FUNCTION_BLOCK fb_V3JRSModuleWithChiller
VAR_INPUT
	bBuiltInTemperetureController : BOOL;
	bBuiltInVacuumSensorController : BOOL;
	bBuiltInVacuumNegativeSignal : BOOL;
END_VAR
VAR_OUTPUT
END_VAR
VAR_IN_OUT
	DS_Alarm :DSV3_JRS_Alarm; (*Channel 200 ~ 204*)
	DS_HMI : DSV3_JRS_HMI; (*Channel of Other Digitial IO and DT*)
	DS_Input : DSV3_JRS_Input; (*Channel 0 ~ 3 *)
	DS_Output : DSV3_JRS_Output; (*Channel 100 ~ 103*)
END_VAR
VAR

	(*Analog Declaration*)
	iThermalOilTempAnalogInput			AT %I* : INT;
	iTopDistillatorTempAnalogInput			AT %I* : INT;
	iBottomDistillatorTempAnalogInput		AT %I* : INT;
	iVaporGenerationTempAnalogInput		AT %I* : INT;
	iColdWaterTankTempAnalogInput 		AT %I* : INT;

	iVacuumSensorAnalogInput				AT %I* : INT;



	(*AlarmControl*)
	arfbTimerAlarm: ARRAY [1..49] OF TIMER_ALARM;
	ARiBuzzerOut : ARRAY [1..4] OF INT;
	ARiAlarmFlag : ARRAY [1..4] OF INT;
	arCMP: ARRAY [1..32] OF CMP_OC_W1;


	(*Others*)
	EQGT: ARRAY [1..10] OF EQ_GT;


	tCompressorOnTimer: TON;
	tCompressorOffTimer: TON;
	tPowerOnDelayTimer: TON;
	tVaporGenTopUpDelayOff: TON;
	tThermalOilChangeResetPBTimer: TON;

	bPowerOnDelay: BOOL;

	t1SecCP: TON;

	tFreshHCCircPumpDelayOffTimer: TON;

	ARtAutoModeTimer: ARRAY [1..4] OF TON;
	ARtManualBoilingTimer: ARRAY [1..4] OF TON;
	diAutoModeDelayTimeSV_Sec: DINT := 20;

	bRecycleStartPBRE: R_TRIG;
	t1SecCPRE: R_TRIG;

	(*Auto BoilDown*)
	t570_AutoBoilingStartDelayTimer: TON;
	t571_AutoBoilDownCompletedDelayTimer: TON;
	t572_AutoBoilSludgeDrainCompletedDelayTimer: TON;
	t573_AutoBoilDistillatorDrainCompletedDelayTimer: TON;
	t574_AutoBoilSludgeDrainCoolingCompletedDelayTimer: TON;        (************* New extra request by customer - YCH************)

	bAutoBoilProcessCompletedFlag: BOOL;
	bAutoBoilDownCompletedFlag: BOOL;
	bAutoBoilSludgeDrainCompletedFlag: BOOL;
	bAutoBoilDistillatorDrainCompletedFlag: BOOL;
	bAutoBoilSludgeDrainCoolingCompletedFlag: BOOL;        (************* New extra request by customer - YCH************)

	(*Manual BoilDown*)
	t590_ManualBoilDownCompletedDelayTimer: TON;
	t591_ManualBoilSludgeCoolingCompletedDelayTimer: TON;
	t592_ManualBoilSludgeDrainCompletedDelayTimer: TON;
	bManualBoilDownCompletedFlag: BOOL;
	bManualBoilSludgeCoolingCompletedFlag: BOOL;
	bManualBoilSludgeDrainCompletedFlag: BOOL;
	bManualBoilSludgeDrainCompletedRE: R_TRIG;
	bManualBoilDownStartPBRE: R_TRIG;

	t592_ManualBoilSludgeDrainCompletedDelayTimerRE: R_TRIG;
	ARfbV2TempControl: ARRAY [1..5] OF fbV2_TempControl;
	rNIL: REAL;

	fbKeyenceVacSensorTuningkPa_Vacuum: fbKeyenceVacSensorTuningkPa;
	bVacuumAchieveFlag: BOOL;

	fbJRSMachine_Routine								: fbV2_EquipmentServiceCounter_Day;
	fbJRSMachine_Major									: fbV2_EquipmentServiceCounter_Day;

	bManulBoilPageOn:BOOL;
(*
	bInternalInput_b000_04_ThermalOilTempCtrlHighTempAlarmSignal : BOOL;
	bInternalInput_b000_05_ThermalOilTempCtrlReadySignal : BOOL;
	bInternalInput_b000_06_ThermalOilTempCtrlOnOffSignal : BOOL;
	bInternalInput_b000_04_ThermalOilTempCtrlHighTempAlarmSignal  : BOOL;
	bInternalInput_b000_05_ThermalOilTempCtrlReadySignal  : BOOL;
	bInternalInput_b000_06_ThermalOilTempCtrlOnOffSignal   : BOOL;

	bInternalInput_b000_07_TopDistillatorTempCtrlHighTempAlarmSignal : BOOL;
	bInternalInput_b000_08_TopDistillatorTempCtrlReadySignal : BOOL;
	bInternalInput_b000_09_TopDistillatorTempCtrlOnOffSignal : BOOL;
	bInternalInput_b000_07_TopDistillatorTempCtrlHighTempAlarmSignal  : BOOL;
	bInternalInput_b000_08_TopDistillatorTempCtrlReadySignal  : BOOL;
	bInternalInput_b000_09_TopDistillatorTempCtrlOnOffSignal   : BOOL;

	bInternalInput_b001_08_BottomDistillatorTempCtrlHighTempAlarmSignal : BOOL;
	bInternalInput_b001_09_BottomDistillatorTempCtrlReadySignal : BOOL;
	bInternalInput_b001_10_BottomDistillatorTempCtrlOnOffSignal : BOOL;
	bInternalInput_b001_08_BottomDistillatorTempCtrlHighTempAlarmSignal  : BOOL;
	bInternalInput_b001_09_BottomDistillatorTempCtrlReadySignal  : BOOL;
	bInternalInput_b001_10_BottomDistillatorTempCtrlOnOffSignal   : BOOL;

	bInternalInput_b002_00_VaporGenerationTempCtrlHighTempAlarmSignal : BOOL;
	bInternalInput_b002_01_VaporGenerationTempCtrlReadySignal : BOOL;
	bInternalInput_b002_02_VaporGenerationTempCtrlOnOffSignal : BOOL;
	bInternalInput_b002_00_VaporGenerationTempCtrlHighTempAlarmSignal  : BOOL;
	bInternalInput_b002_01_VaporGenerationTempCtrlReadySignal  : BOOL;
	bInternalInput_b002_02_VaporGenerationTempCtrlOnOffSignal  : BOOL;


	bInternalInput_b003_03_ColdWaterTankTempCtrlHighTempAlarmSignal : BOOL;
	bInternalInput_b003_04_ColdWaterTankTempCtrlReadySignal : BOOL;
	bInternalInput_b003_05_ColdWaterTankTempCtrlOnOffSignal	 : BOOL;
	bInternalInput_b003_03_ColdWaterTankTempCtrlHighTempAlarmSignal  : BOOL;
	bInternalInput_b003_04_ColdWaterTankTempCtrlReadySignal  : BOOL;
	bInternalInput_b003_05_ColdWaterTankTempCtrlOnOffSignal  : BOOL;

	bInternalInput_b001_04_VacuumNotAchieveSignal	: BOOL;
	bInternalInput_b001_04_VacuumNotAchieveSignal  : BOOL;

*)

	(*Internal Signal Declaration*)
	bInternalAlarm_b200_00_FreshHCTankCircPumpTORAlarm   : BOOL;
	bInternalAlarm_b200_01_CircTankCircPumpTORAlarm   : BOOL;
	bInternalAlarm_b200_02_ThermalOilPumpTORAlarm   : BOOL;
	bInternalAlarm_b200_03_ThermalOilLowLevelAlarm   : BOOL;
	bInternalAlarm_b200_04_ThermalOilTempHighAlarm   : BOOL;
	bInternalAlarm_b200_05_ThermalOilTempNotReadyAlarm   : BOOL;
	bInternalAlarm_b200_06_ThermalOilHeaterOnOffAlarm   : BOOL;
	bInternalAlarm_b200_07_TopDistillatorTempHighAlarm   : BOOL;
	bInternalAlarm_b200_08_TopDistillatorTempNotReadyAlarm   : BOOL;
	bInternalAlarm_b200_09_TopDistillatorHeaterOnOffAlarm   : BOOL;
	bInternalAlarm_b200_10_RecycleStartStopPBAlarm   : BOOL;
	bInternalAlarm_b200_11_EstopPBAlarm   : BOOL;

	bInternalAlarm_b201_00_PhaseSeqenceRelayAlarm   : BOOL;
	bInternalAlarm_b201_01_ThermalOilUpThermostatAlarm   : BOOL;
	bInternalAlarm_b201_02_SludgeTankHighLevelAlarm   : BOOL;
	bInternalAlarm_b201_03_FreshHCTankLowLevelAlarm   : BOOL;
	bInternalAlarm_b201_04_VacuumNotAchieveAlarm   : BOOL;
	bInternalAlarm_b201_05_IncomingCDALowPressureAlarm   : BOOL;
	bInternalAlarm_b201_06_CoolingWaterLowFlowAlarm   : BOOL;
	bInternalAlarm_b201_07_CircularTankLowLevelAlarm   : BOOL;
	bInternalAlarm_b201_08_BottomDistillatorTempHighAlarm   : BOOL;
	bInternalAlarm_b201_09_BottomDistillatorTempNotReadyAlarm   : BOOL;
	bInternalAlarm_b201_10_BottomDistillatorHeaterOnOffAlarm   : BOOL;
	bInternalAlarm_b201_11_ThermalOilDownThermostatAlarm   : BOOL;
	bInternalAlarm_b201_12_ThermalOilMidThermostatAlarm   : BOOL;

	bInternalAlarm_b202_00_VaporGenerationTempHighAlarm   : BOOL;
	bInternalAlarm_b202_01_VaporGenerationTempNotReadyAlarm   : BOOL;
	bInternalAlarm_b202_02_VaporGenerationHeaterOnOffAlarm   : BOOL;
	bInternalAlarm_b202_03_WasteCollectionTankLowLevelAlarm   : BOOL;
	bInternalAlarm_b202_04_VaporGenerationTankLowLevelAlarm   : BOOL;
	bInternalAlarm_b202_05_HCPurgingAV3_1Alarm   : BOOL;
	bInternalAlarm_b202_06_MainMachineWasteTankLowLevelAlarm   : BOOL;
	bInternalAlarm_b202_07_MainMachineWasteTankHighLevelAlarm   : BOOL;
	bInternalAlarm_b202_08_ReservedAlarm   : BOOL;
	bInternalAlarm_b202_09_ReservedAlarm   : BOOL;
	bInternalAlarm_b202_10_ReservedAlarm   : BOOL;
	bInternalAlarm_b202_11_ReservedAlarm   : BOOL;

	bInternalAlarm_b203_00_ChillerSelectorOnOffAlarm   : BOOL;
	bInternalAlarm_b203_01_ColdWaterTankLowLevelAlarm   : BOOL;
	bInternalAlarm_b203_02_SludgeTankMissingAlarm   : BOOL;
	bInternalAlarm_b203_03_ColdWaterTankTempHighAlarm   : BOOL;
	bInternalAlarm_b203_04_ColdWaterTankTempNotReadyAlarm   : BOOL;
	bInternalAlarm_b203_05_ColdWaterTankHeaterOnOffAlarm   : BOOL;
	bInternalAlarm_b203_06_ChillerPumpTORAlarm   : BOOL;
	bInternalAlarm_b203_07_ChillerFlowSwitchAlarm   : BOOL;
	bInternalAlarm_b203_08_ChillerInterlockRelayAlarm   : BOOL;
	bInternalAlarm_b203_09_ReservedAlarm   : BOOL;
	bInternalAlarm_b203_10_ThermalOilChangeWarning   : BOOL;
	bInternalAlarm_b203_11_ThermalOilChangeAlarm   : BOOL;



	bInternalInput_b000_00_FreshHCTankCircPumpTOR   : BOOL;
	bInternalInput_b000_01_CircTankCircPumpTOR   : BOOL;
	bInternalInput_b000_02_ThermalOilPumpTOR  : BOOL;
	bInternalInput_b000_03_ThermalOilLevelSensor  : BOOL;
	bInternalInput_b000_04_ThermalOilTempCtrlHighTempAlarmSignal  : BOOL;
	bInternalInput_b000_05_ThermalOilTempCtrlReadySignal  : BOOL;
	bInternalInput_b000_06_ThermalOilTempCtrlOnOffSignal   : BOOL;
	bInternalInput_b000_07_TopDistillatorTempCtrlHighTempAlarmSignal  : BOOL;
	bInternalInput_b000_08_TopDistillatorTempCtrlReadySignal  : BOOL;
	bInternalInput_b000_09_TopDistillatorTempCtrlOnOffSignal   : BOOL;
	bInternalInput_b000_10_RecycleStartStopPB  : BOOL;
	bInternalInput_b000_11_EStopPB  : BOOL;


	bInternalInput_b001_00_PhaseSequenceRelayAlarm  : BOOL;
	bInternalInput_b001_01_ThermalOilUpThermostat   : BOOL;
	bInternalInput_b001_02_SludgeTankLevelSensor  : BOOL;
	bInternalInput_b001_03_FreshHCTankLevelSensor  : BOOL;
	bInternalInput_b001_04_VacuumNotAchieveSignal  : BOOL;
	bInternalInput_b001_05_IncomingCDAPressureSwitch  : BOOL;
	bInternalInput_b001_06_CoolingWaterFlowSwitch  : BOOL;
	bInternalInput_b001_07_CircularTankLevelSensor  : BOOL;
	bInternalInput_b001_08_BottomDistillatorTempCtrlHighTempAlarmSignal  : BOOL;
	bInternalInput_b001_09_BottomDistillatorTempCtrlReadySignal  : BOOL;
	bInternalInput_b001_10_BottomDistillatorTempCtrlOnOffSignal   : BOOL;
	bInternalInput_b001_11_ThermalOilDownThermostat  : BOOL;
	bInternalInput_b001_12_ThermalOilMidThermostat  : BOOL;

	bInternalInput_b002_00_VaporGenerationTempCtrlHighTempAlarmSignal  : BOOL;
	bInternalInput_b002_01_VaporGenerationTempCtrlReadySignal  : BOOL;
	bInternalInput_b002_02_VaporGenerationTempCtrlOnOffSignal  : BOOL;
	bInternalInput_b002_03_WasteCollectionTankLevelSensor  : BOOL;
	bInternalInput_b002_04_VaporGenerationTankLowLevelSensor  : BOOL;
	bInternalInput_b002_05_HCPurgingAV  : BOOL;
	bInternalInput_b002_06_MainMachineWasteCollectTankLowLevelSignal  : BOOL;
	bInternalInput_b002_07_MainMachineWasteCollectTankHighLevelSignal  : BOOL;
	bInternalInput_b002_08_FromMainMachineSignal3  : BOOL;
	bInternalInput_b002_09_FromMainMachineSignal4  : BOOL;
	bInternalInput_b002_10_FromMainMachineSignal5  : BOOL;
	bInternalInput_b002_11_ReservedAlarmSignal  : BOOL;


	bInternalInput_b003_00_ChillerSelectorOnOff  : BOOL;
	bInternalInput_b003_01_ColdWaterTankLowLevelSensor  : BOOL;
	bInternalInput_b003_02_SludgeTankPresentSensor  : BOOL;
	bInternalInput_b003_03_ColdWaterTankTempCtrlHighTempAlarmSignal  : BOOL;
	bInternalInput_b003_04_ColdWaterTankTempCtrlReadySignal  : BOOL;
	bInternalInput_b003_05_ColdWaterTankTempCtrlOnOffSignal  : BOOL;
	bInternalInput_b003_06_ChillerPumpTOR  : BOOL;
	bInternalInput_b003_07_ChillerFlowSwitch  : BOOL;
	bInternalInput_b003_08_ChillerInterlockRelay  : BOOL;
	bInternalInput_b003_09_ReservedAlarmSignal  : BOOL;
	bInternalInput_b003_10_ReservedAlarmSignal  : BOOL;
	bInternalInput_b003_11_ReservedAlarmSignal  : BOOL;


	bInternalOutput_b100_00_FreshHCTankCircPumpOnOff   : BOOL;
	bInternalOutput_b100_01_CircTankCircPumpOnOff  : BOOL;
	bInternalOutput_b100_02_ThermalOilPumpOnOff  : BOOL;
	bInternalOutput_b100_03_ThermalOilHeaterOnOff  : BOOL;
	bInternalOutput_b100_04_Buzzer  : BOOL;
	bInternalOutput_b100_05_RecycleStartStopIndicator  : BOOL;
	bInternalOutput_b100_06_Reserved  : BOOL;
	bInternalOutput_b100_07_UFOVacuumRelease32WayAV  : BOOL;


	bInternalOutput_b101_00_CondenserTankVacuumReleaseAV  : BOOL;
	bInternalOutput_b101_01_WasteSludgeCollectionDrumAV   : BOOL;
	bInternalOutput_b101_02_DistillationTankDrainAV  : BOOL;
	bInternalOutput_b101_03_EconomizerAV  : BOOL;
	bInternalOutput_b101_04_Reserved  : BOOL;
	bInternalOutput_b101_05_Reserved  : BOOL;
	bInternalOutput_b101_06_VaporGenerationAV  : BOOL;
	bInternalOutput_b101_07_VacuumSharingAV  : BOOL;


	bInternalOutput_b102_00_RecycleReadySignal  : BOOL;
	bInternalOutput_b102_01_VaporNotAvailableForRequestSignal  : BOOL;
	bInternalOutput_b102_02_ToMainMachineSignal3  : BOOL;
	bInternalOutput_b102_03_ToMainMachineSignal4  : BOOL;
	bInternalOutput_b102_04_ToMainMachineSignal5  : BOOL;
	bInternalOutput_b102_05_Reserved  : BOOL;
	bInternalOutput_b102_06_Reserved  : BOOL;
	bInternalOutput_b102_07_Reserved  : BOOL;


	bInternalOutput_b103_00_ChillerPumpOnOff  : BOOL;
	bInternalOutput_b103_01_Reserved  : BOOL;
	bInternalOutput_b103_02_Reserved  : BOOL;
	bInternalOutput_b103_03_Reserved  : BOOL;
	bInternalOutput_b103_04_ChillerSelectorOnOffIndicator  : BOOL;
	bInternalOutput_b103_05_ChillerReadySignal  : BOOL;
	bInternalOutput_b103_06_ChillerCompressorOnOff  : BOOL;
	bInternalOutput_b103_07_Reserved  : BOOL;


END_VAR
VAR // added by the converter: edge detectors and wires of the graphical bodies
    _w1, _w3, _w4, _w5, _w6, _w7, _w8, _w9 : ANY;
    _w2 : BOOL;
END_VAR

	(*Timer*)
	t1SecCP(IN:=NOT t1SecCP.Q , PT:=t#1s , Q=> , ET=> );


	(*R_TRIG*)
	t1SecCPRE(CLK:=t1SecCP.Q , Q=> );
	bRecycleStartPBRE(CLK:=bInternalInput_b000_10_RecycleStartStopPB , Q=> );


	(*Sub Program Execution*)
	Z_Mapping();
	Other_LD();
	Other_ST();
	FixOutput_LD();
	OutputCtrl_LD();
	AlarmCtrl_LD();
	BuzzerCtrl_ST();
	MessageDisplayCtrl_ST();
	AutoHCTopUp_LD();
	HighLowLimitCtrl_ST();
	AutoCtrl_LD();
	ManualCtrl_ST();
	
	AutoBoilingCtrl_LD();
	AutoBoilingCtrl_ST();

	ManualBoilingCtrl_LD();
	ManualBoilingCtrl_ST();


	ThermalOilChangeHRMeter_ST();
	ChillerCtrl_LD();
	SystemRestore_LD();
	Z_BuiltInTempCtrl_ST();

	Z_BuiltInVacuumCtrl_ST();

	JRSMachineServiceCtrl_LD();

ACTION AlarmCtrl_LD:
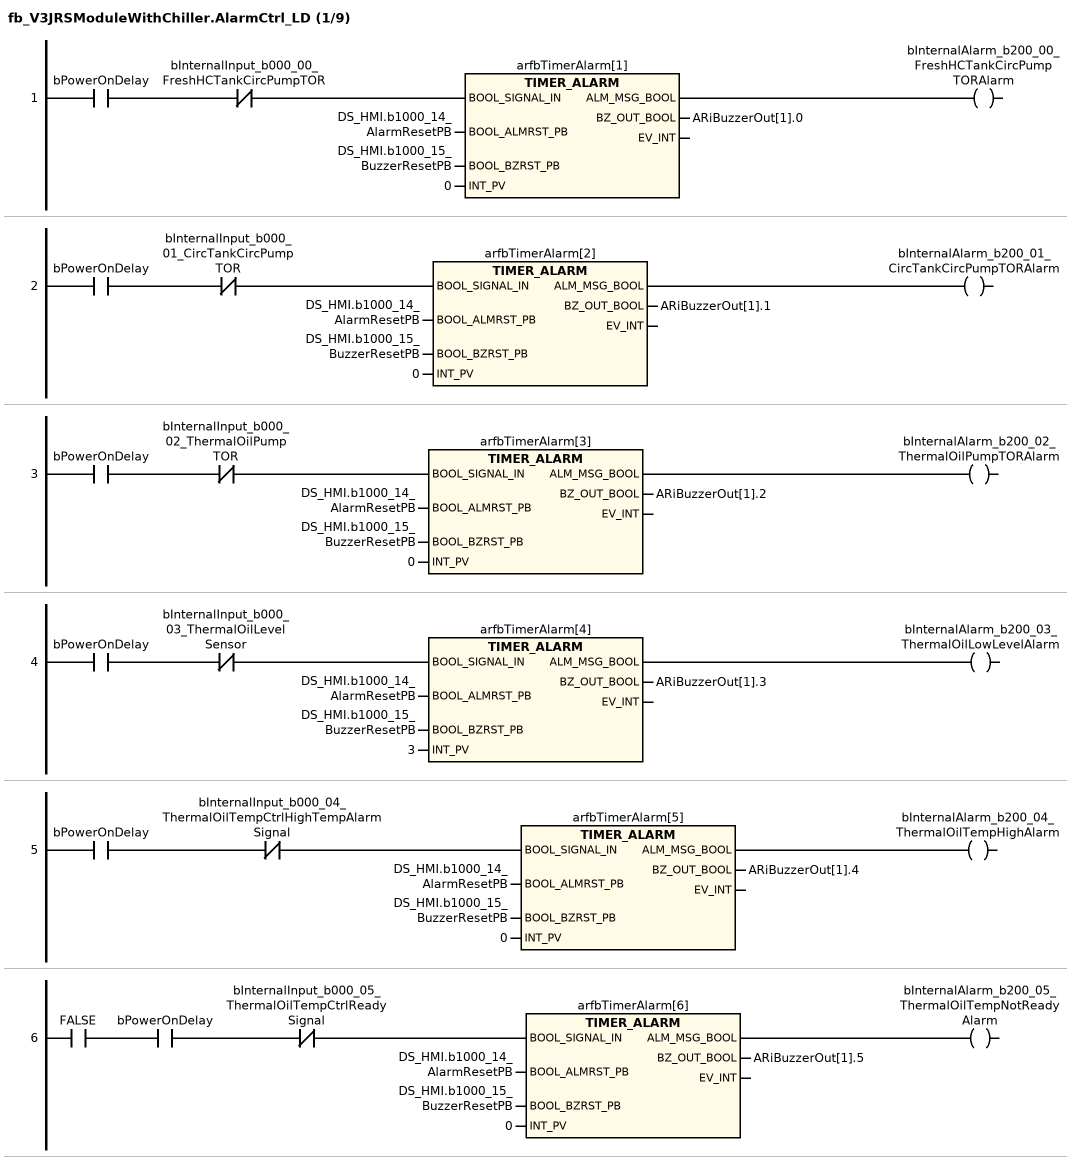
// NETWORK 1
arfbTimerAlarm[1](
    BOOL_SIGNAL_IN := bPowerOnDelay AND NOT bInternalInput_b000_00_FreshHCTankCircPumpTOR,
    BOOL_ALMRST_PB := DS_HMI.b1000_14_AlarmResetPB,
    BOOL_BZRST_PB := DS_HMI.b1000_15_BuzzerResetPB,
    INT_PV := 0,
    BZ_OUT_BOOL => ARiBuzzerOut[1].0); // TIMER_ALARM
bInternalAlarm_b200_00_FreshHCTankCircPumpTORAlarm := arfbTimerAlarm[1].ALM_MSG_BOOL;

// NETWORK 2
arfbTimerAlarm[2](
    BOOL_SIGNAL_IN := bPowerOnDelay AND NOT bInternalInput_b000_01_CircTankCircPumpTOR,
    BOOL_ALMRST_PB := DS_HMI.b1000_14_AlarmResetPB,
    BOOL_BZRST_PB := DS_HMI.b1000_15_BuzzerResetPB,
    INT_PV := 0,
    BZ_OUT_BOOL => ARiBuzzerOut[1].1); // TIMER_ALARM
bInternalAlarm_b200_01_CircTankCircPumpTORAlarm := arfbTimerAlarm[2].ALM_MSG_BOOL;

// NETWORK 3
arfbTimerAlarm[3](
    BOOL_SIGNAL_IN := bPowerOnDelay AND NOT bInternalInput_b000_02_ThermalOilPumpTOR,
    BOOL_ALMRST_PB := DS_HMI.b1000_14_AlarmResetPB,
    BOOL_BZRST_PB := DS_HMI.b1000_15_BuzzerResetPB,
    INT_PV := 0,
    BZ_OUT_BOOL => ARiBuzzerOut[1].2); // TIMER_ALARM
bInternalAlarm_b200_02_ThermalOilPumpTORAlarm := arfbTimerAlarm[3].ALM_MSG_BOOL;

// NETWORK 4
arfbTimerAlarm[4](
    BOOL_SIGNAL_IN := bPowerOnDelay AND NOT bInternalInput_b000_03_ThermalOilLevelSensor,
    BOOL_ALMRST_PB := DS_HMI.b1000_14_AlarmResetPB,
    BOOL_BZRST_PB := DS_HMI.b1000_15_BuzzerResetPB,
    INT_PV := 3,
    BZ_OUT_BOOL => ARiBuzzerOut[1].3); // TIMER_ALARM
bInternalAlarm_b200_03_ThermalOilLowLevelAlarm := arfbTimerAlarm[4].ALM_MSG_BOOL;

// NETWORK 5
arfbTimerAlarm[5](
    BOOL_SIGNAL_IN := bPowerOnDelay AND NOT bInternalInput_b000_04_ThermalOilTempCtrlHighTempAlarmSignal,
    BOOL_ALMRST_PB := DS_HMI.b1000_14_AlarmResetPB,
    BOOL_BZRST_PB := DS_HMI.b1000_15_BuzzerResetPB,
    INT_PV := 0,
    BZ_OUT_BOOL => ARiBuzzerOut[1].4); // TIMER_ALARM
bInternalAlarm_b200_04_ThermalOilTempHighAlarm := arfbTimerAlarm[5].ALM_MSG_BOOL;

// NETWORK 6
arfbTimerAlarm[6](
    BOOL_SIGNAL_IN := FALSE AND bPowerOnDelay AND NOT bInternalInput_b000_05_ThermalOilTempCtrlReadySignal,
    BOOL_ALMRST_PB := DS_HMI.b1000_14_AlarmResetPB,
    BOOL_BZRST_PB := DS_HMI.b1000_15_BuzzerResetPB,
    INT_PV := 0,
    BZ_OUT_BOOL => ARiBuzzerOut[1].5); // TIMER_ALARM
bInternalAlarm_b200_05_ThermalOilTempNotReadyAlarm := arfbTimerAlarm[6].ALM_MSG_BOOL;

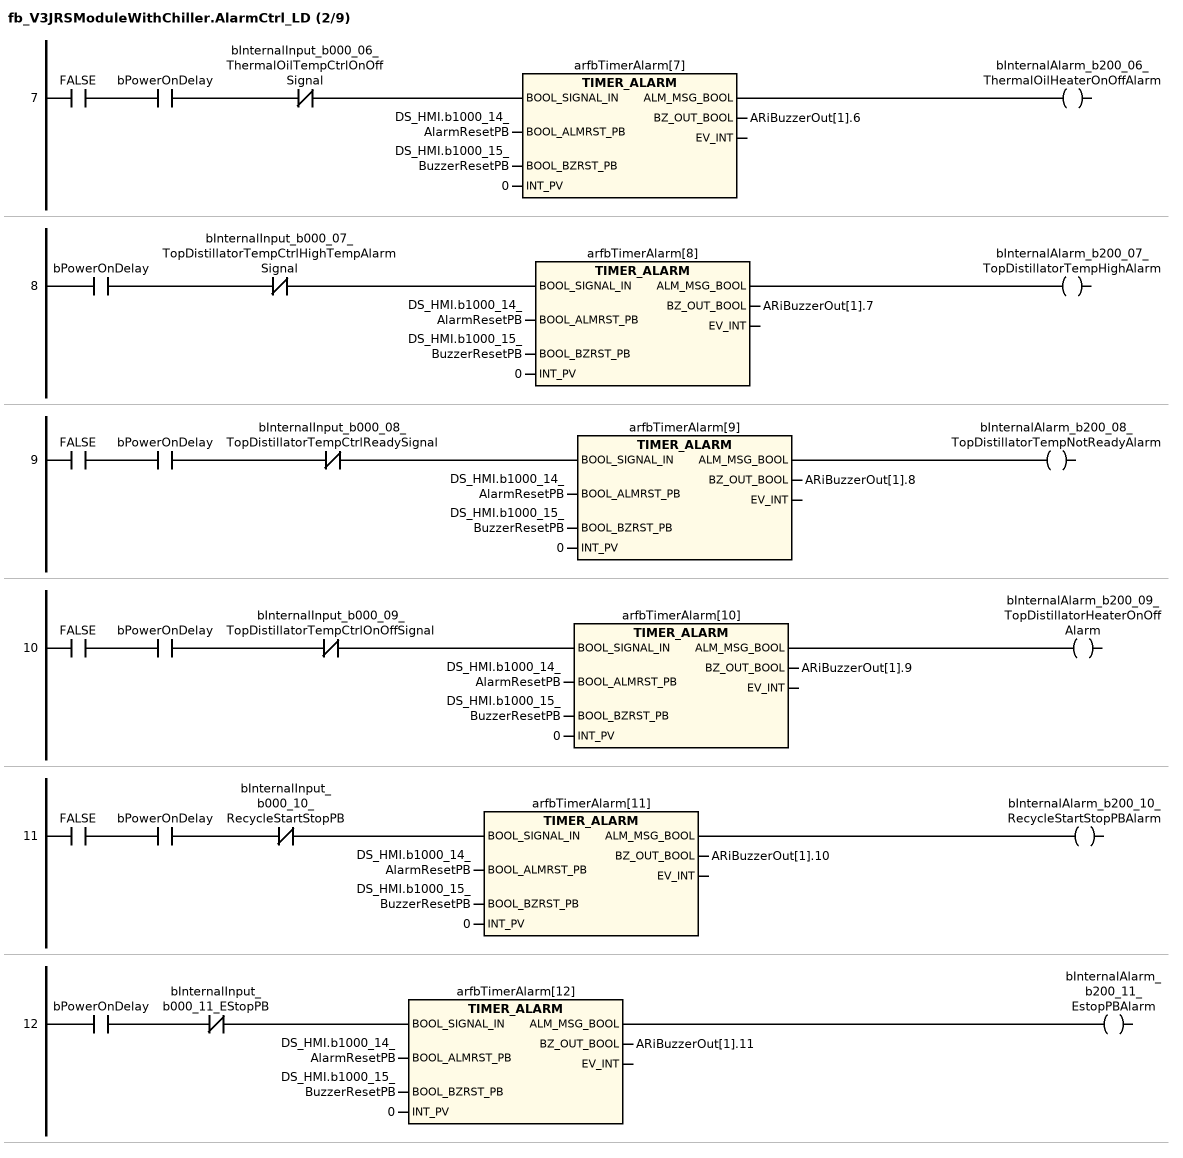
// NETWORK 7
arfbTimerAlarm[7](
    BOOL_SIGNAL_IN := FALSE AND bPowerOnDelay AND NOT bInternalInput_b000_06_ThermalOilTempCtrlOnOffSignal,
    BOOL_ALMRST_PB := DS_HMI.b1000_14_AlarmResetPB,
    BOOL_BZRST_PB := DS_HMI.b1000_15_BuzzerResetPB,
    INT_PV := 0,
    BZ_OUT_BOOL => ARiBuzzerOut[1].6); // TIMER_ALARM
bInternalAlarm_b200_06_ThermalOilHeaterOnOffAlarm := arfbTimerAlarm[7].ALM_MSG_BOOL;

// NETWORK 8
arfbTimerAlarm[8](
    BOOL_SIGNAL_IN := bPowerOnDelay AND NOT bInternalInput_b000_07_TopDistillatorTempCtrlHighTempAlarmSignal,
    BOOL_ALMRST_PB := DS_HMI.b1000_14_AlarmResetPB,
    BOOL_BZRST_PB := DS_HMI.b1000_15_BuzzerResetPB,
    INT_PV := 0,
    BZ_OUT_BOOL => ARiBuzzerOut[1].7); // TIMER_ALARM
bInternalAlarm_b200_07_TopDistillatorTempHighAlarm := arfbTimerAlarm[8].ALM_MSG_BOOL;

// NETWORK 9
arfbTimerAlarm[9](
    BOOL_SIGNAL_IN := FALSE AND bPowerOnDelay AND NOT bInternalInput_b000_08_TopDistillatorTempCtrlReadySignal,
    BOOL_ALMRST_PB := DS_HMI.b1000_14_AlarmResetPB,
    BOOL_BZRST_PB := DS_HMI.b1000_15_BuzzerResetPB,
    INT_PV := 0,
    BZ_OUT_BOOL => ARiBuzzerOut[1].8); // TIMER_ALARM
bInternalAlarm_b200_08_TopDistillatorTempNotReadyAlarm := arfbTimerAlarm[9].ALM_MSG_BOOL;

// NETWORK 10
arfbTimerAlarm[10](
    BOOL_SIGNAL_IN := FALSE AND bPowerOnDelay AND NOT bInternalInput_b000_09_TopDistillatorTempCtrlOnOffSignal,
    BOOL_ALMRST_PB := DS_HMI.b1000_14_AlarmResetPB,
    BOOL_BZRST_PB := DS_HMI.b1000_15_BuzzerResetPB,
    INT_PV := 0,
    BZ_OUT_BOOL => ARiBuzzerOut[1].9); // TIMER_ALARM
bInternalAlarm_b200_09_TopDistillatorHeaterOnOffAlarm := arfbTimerAlarm[10].ALM_MSG_BOOL;

// NETWORK 11
arfbTimerAlarm[11](
    BOOL_SIGNAL_IN := FALSE AND bPowerOnDelay AND NOT bInternalInput_b000_10_RecycleStartStopPB,
    BOOL_ALMRST_PB := DS_HMI.b1000_14_AlarmResetPB,
    BOOL_BZRST_PB := DS_HMI.b1000_15_BuzzerResetPB,
    INT_PV := 0,
    BZ_OUT_BOOL => ARiBuzzerOut[1].10); // TIMER_ALARM
bInternalAlarm_b200_10_RecycleStartStopPBAlarm := arfbTimerAlarm[11].ALM_MSG_BOOL;

// NETWORK 12
arfbTimerAlarm[12](
    BOOL_SIGNAL_IN := bPowerOnDelay AND NOT bInternalInput_b000_11_EStopPB,
    BOOL_ALMRST_PB := DS_HMI.b1000_14_AlarmResetPB,
    BOOL_BZRST_PB := DS_HMI.b1000_15_BuzzerResetPB,
    INT_PV := 0,
    BZ_OUT_BOOL => ARiBuzzerOut[1].11); // TIMER_ALARM
bInternalAlarm_b200_11_EstopPBAlarm := arfbTimerAlarm[12].ALM_MSG_BOOL;

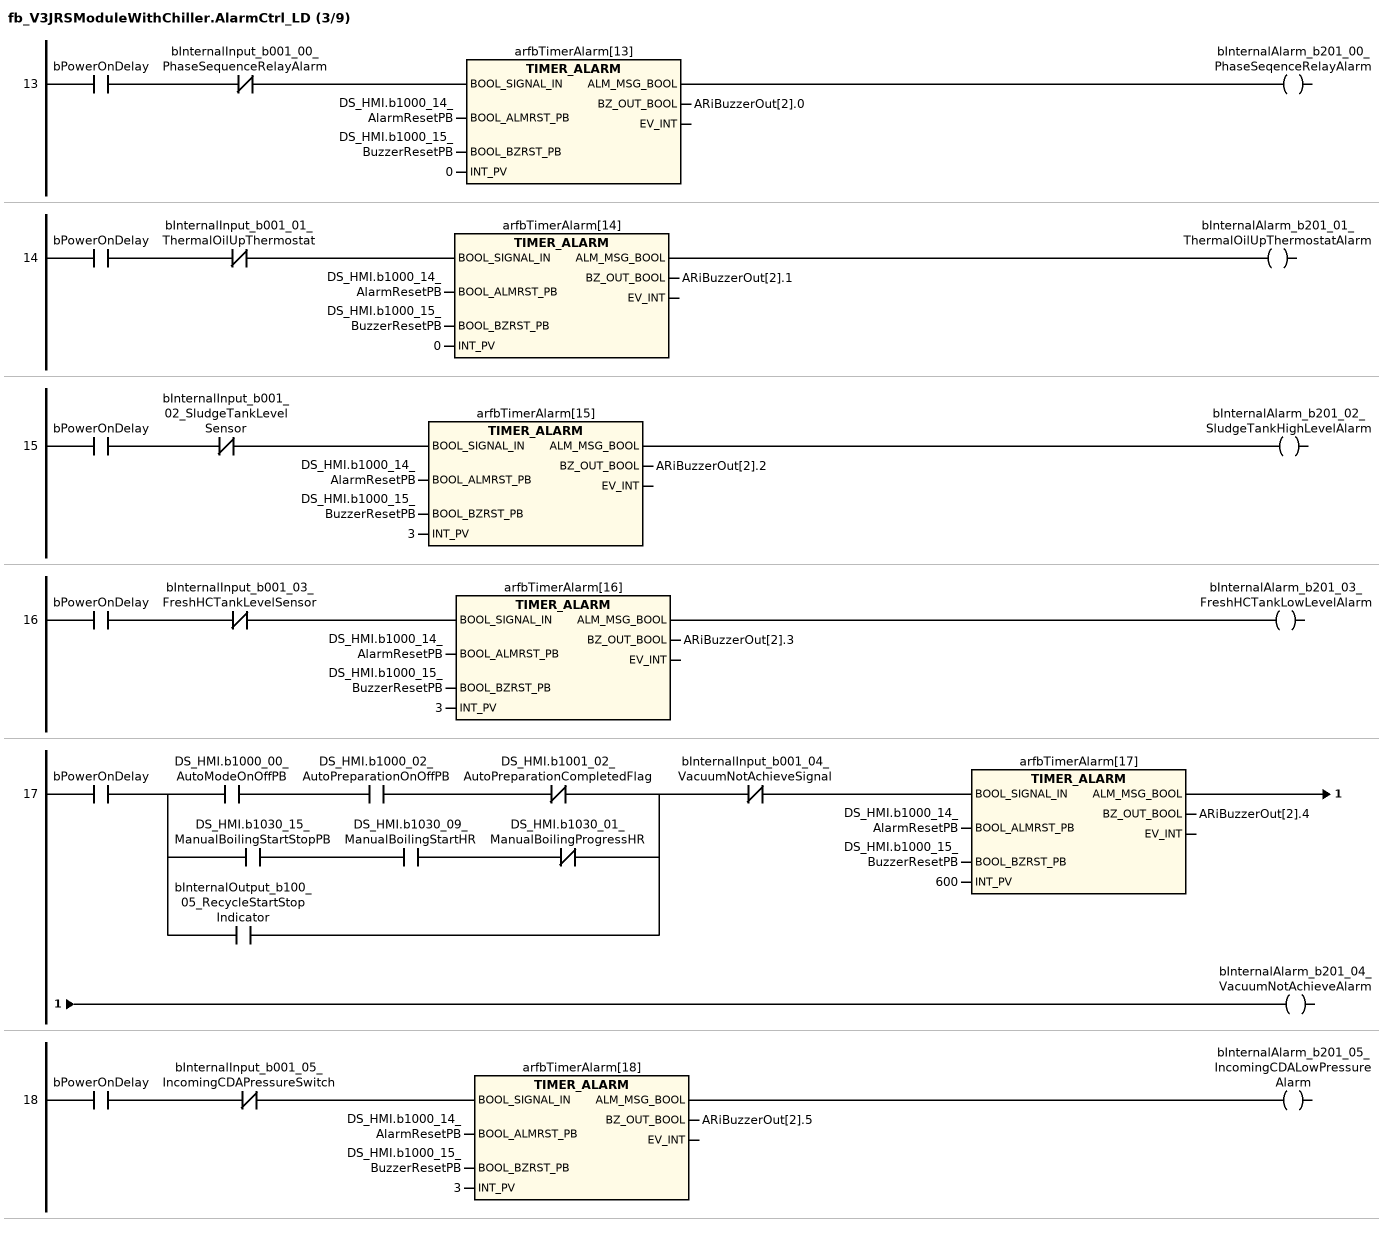
// NETWORK 13
arfbTimerAlarm[13](
    BOOL_SIGNAL_IN := bPowerOnDelay AND NOT bInternalInput_b001_00_PhaseSequenceRelayAlarm,
    BOOL_ALMRST_PB := DS_HMI.b1000_14_AlarmResetPB,
    BOOL_BZRST_PB := DS_HMI.b1000_15_BuzzerResetPB,
    INT_PV := 0,
    BZ_OUT_BOOL => ARiBuzzerOut[2].0); // TIMER_ALARM
bInternalAlarm_b201_00_PhaseSeqenceRelayAlarm := arfbTimerAlarm[13].ALM_MSG_BOOL;

// NETWORK 14
arfbTimerAlarm[14](
    BOOL_SIGNAL_IN := bPowerOnDelay AND NOT bInternalInput_b001_01_ThermalOilUpThermostat,
    BOOL_ALMRST_PB := DS_HMI.b1000_14_AlarmResetPB,
    BOOL_BZRST_PB := DS_HMI.b1000_15_BuzzerResetPB,
    INT_PV := 0,
    BZ_OUT_BOOL => ARiBuzzerOut[2].1); // TIMER_ALARM
bInternalAlarm_b201_01_ThermalOilUpThermostatAlarm := arfbTimerAlarm[14].ALM_MSG_BOOL;

// NETWORK 15
arfbTimerAlarm[15](
    BOOL_SIGNAL_IN := bPowerOnDelay AND NOT bInternalInput_b001_02_SludgeTankLevelSensor,
    BOOL_ALMRST_PB := DS_HMI.b1000_14_AlarmResetPB,
    BOOL_BZRST_PB := DS_HMI.b1000_15_BuzzerResetPB,
    INT_PV := 3,
    BZ_OUT_BOOL => ARiBuzzerOut[2].2); // TIMER_ALARM
bInternalAlarm_b201_02_SludgeTankHighLevelAlarm := arfbTimerAlarm[15].ALM_MSG_BOOL;

// NETWORK 16
arfbTimerAlarm[16](
    BOOL_SIGNAL_IN := bPowerOnDelay AND NOT bInternalInput_b001_03_FreshHCTankLevelSensor,
    BOOL_ALMRST_PB := DS_HMI.b1000_14_AlarmResetPB,
    BOOL_BZRST_PB := DS_HMI.b1000_15_BuzzerResetPB,
    INT_PV := 3,
    BZ_OUT_BOOL => ARiBuzzerOut[2].3); // TIMER_ALARM
bInternalAlarm_b201_03_FreshHCTankLowLevelAlarm := arfbTimerAlarm[16].ALM_MSG_BOOL;

// NETWORK 17
arfbTimerAlarm[17](
    BOOL_SIGNAL_IN := (bPowerOnDelay AND (DS_HMI.b1000_00_AutoModeOnOffPB AND DS_HMI.b1000_02_AutoPreparationOnOffPB AND NOT DS_HMI.b1001_02_AutoPreparationCompletedFlag OR DS_HMI.b1030_15_ManualBoilingStartStopPB AND DS_HMI.b1030_09_ManualBoilingStartHR AND NOT DS_HMI.b1030_01_ManualBoilingProgressHR OR bInternalOutput_b100_05_RecycleStartStopIndicator)) AND NOT bInternalInput_b001_04_VacuumNotAchieveSignal,
    BOOL_ALMRST_PB := DS_HMI.b1000_14_AlarmResetPB,
    BOOL_BZRST_PB := DS_HMI.b1000_15_BuzzerResetPB,
    INT_PV := 600,
    BZ_OUT_BOOL => ARiBuzzerOut[2].4); // TIMER_ALARM
bInternalAlarm_b201_04_VacuumNotAchieveAlarm := arfbTimerAlarm[17].ALM_MSG_BOOL;

// NETWORK 18
arfbTimerAlarm[18](
    BOOL_SIGNAL_IN := bPowerOnDelay AND NOT bInternalInput_b001_05_IncomingCDAPressureSwitch,
    BOOL_ALMRST_PB := DS_HMI.b1000_14_AlarmResetPB,
    BOOL_BZRST_PB := DS_HMI.b1000_15_BuzzerResetPB,
    INT_PV := 3,
    BZ_OUT_BOOL => ARiBuzzerOut[2].5); // TIMER_ALARM
bInternalAlarm_b201_05_IncomingCDALowPressureAlarm := arfbTimerAlarm[18].ALM_MSG_BOOL;

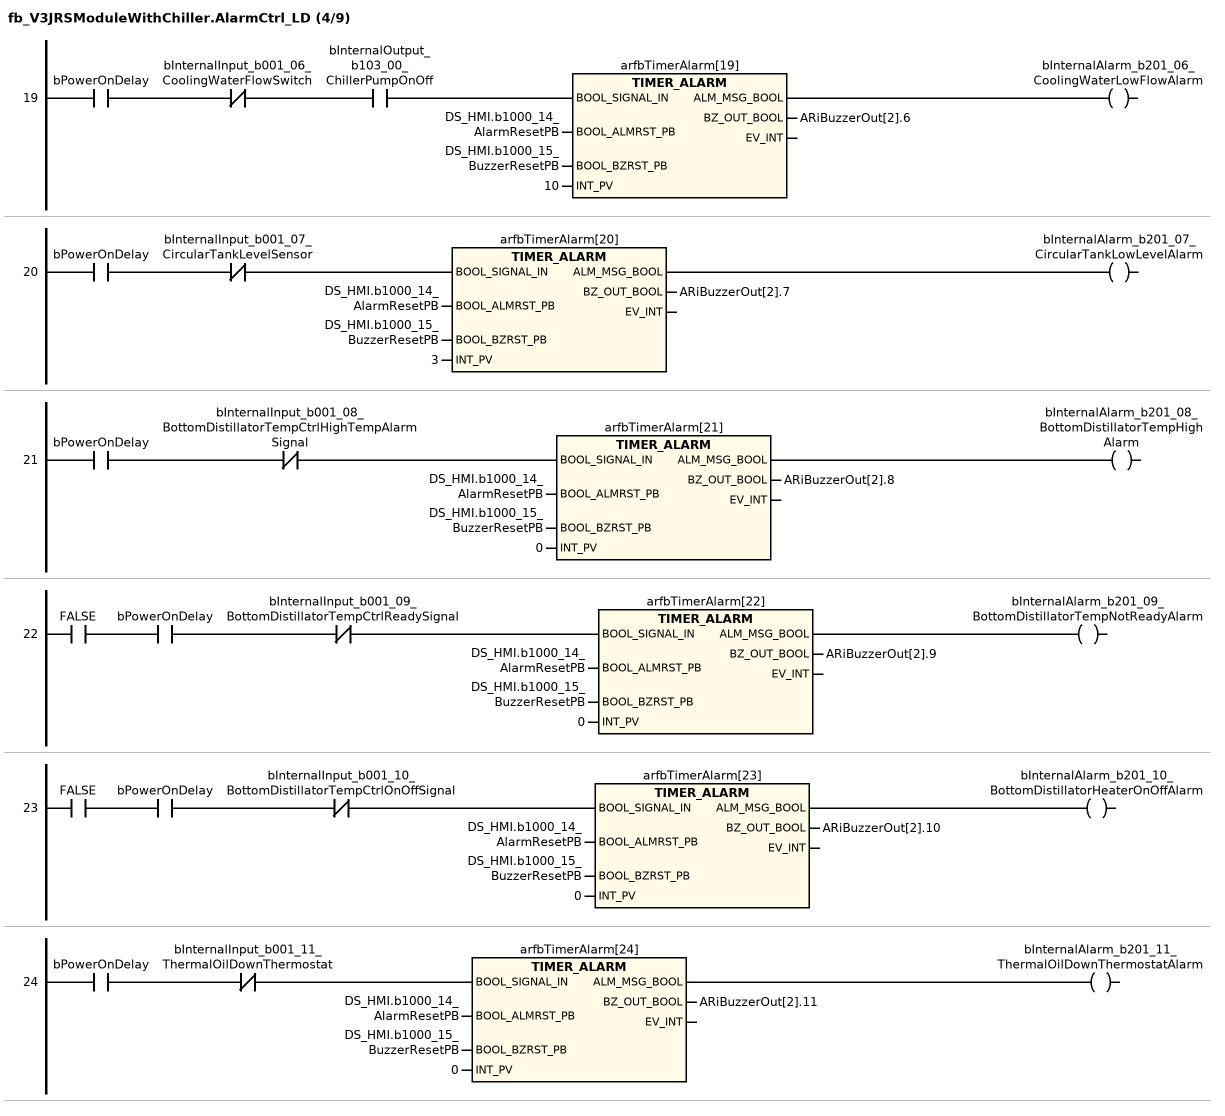
// NETWORK 19
arfbTimerAlarm[19](
    BOOL_SIGNAL_IN := bPowerOnDelay AND NOT bInternalInput_b001_06_CoolingWaterFlowSwitch AND bInternalOutput_b103_00_ChillerPumpOnOff,
    BOOL_ALMRST_PB := DS_HMI.b1000_14_AlarmResetPB,
    BOOL_BZRST_PB := DS_HMI.b1000_15_BuzzerResetPB,
    INT_PV := 10,
    BZ_OUT_BOOL => ARiBuzzerOut[2].6); // TIMER_ALARM
bInternalAlarm_b201_06_CoolingWaterLowFlowAlarm := arfbTimerAlarm[19].ALM_MSG_BOOL;

// NETWORK 20
arfbTimerAlarm[20](
    BOOL_SIGNAL_IN := bPowerOnDelay AND NOT bInternalInput_b001_07_CircularTankLevelSensor,
    BOOL_ALMRST_PB := DS_HMI.b1000_14_AlarmResetPB,
    BOOL_BZRST_PB := DS_HMI.b1000_15_BuzzerResetPB,
    INT_PV := 3,
    BZ_OUT_BOOL => ARiBuzzerOut[2].7); // TIMER_ALARM
bInternalAlarm_b201_07_CircularTankLowLevelAlarm := arfbTimerAlarm[20].ALM_MSG_BOOL;

// NETWORK 21
arfbTimerAlarm[21](
    BOOL_SIGNAL_IN := bPowerOnDelay AND NOT bInternalInput_b001_08_BottomDistillatorTempCtrlHighTempAlarmSignal,
    BOOL_ALMRST_PB := DS_HMI.b1000_14_AlarmResetPB,
    BOOL_BZRST_PB := DS_HMI.b1000_15_BuzzerResetPB,
    INT_PV := 0,
    BZ_OUT_BOOL => ARiBuzzerOut[2].8); // TIMER_ALARM
bInternalAlarm_b201_08_BottomDistillatorTempHighAlarm := arfbTimerAlarm[21].ALM_MSG_BOOL;

// NETWORK 22
arfbTimerAlarm[22](
    BOOL_SIGNAL_IN := FALSE AND bPowerOnDelay AND NOT bInternalInput_b001_09_BottomDistillatorTempCtrlReadySignal,
    BOOL_ALMRST_PB := DS_HMI.b1000_14_AlarmResetPB,
    BOOL_BZRST_PB := DS_HMI.b1000_15_BuzzerResetPB,
    INT_PV := 0,
    BZ_OUT_BOOL => ARiBuzzerOut[2].9); // TIMER_ALARM
bInternalAlarm_b201_09_BottomDistillatorTempNotReadyAlarm := arfbTimerAlarm[22].ALM_MSG_BOOL;

// NETWORK 23
arfbTimerAlarm[23](
    BOOL_SIGNAL_IN := FALSE AND bPowerOnDelay AND NOT bInternalInput_b001_10_BottomDistillatorTempCtrlOnOffSignal,
    BOOL_ALMRST_PB := DS_HMI.b1000_14_AlarmResetPB,
    BOOL_BZRST_PB := DS_HMI.b1000_15_BuzzerResetPB,
    INT_PV := 0,
    BZ_OUT_BOOL => ARiBuzzerOut[2].10); // TIMER_ALARM
bInternalAlarm_b201_10_BottomDistillatorHeaterOnOffAlarm := arfbTimerAlarm[23].ALM_MSG_BOOL;

// NETWORK 24
arfbTimerAlarm[24](
    BOOL_SIGNAL_IN := bPowerOnDelay AND NOT bInternalInput_b001_11_ThermalOilDownThermostat,
    BOOL_ALMRST_PB := DS_HMI.b1000_14_AlarmResetPB,
    BOOL_BZRST_PB := DS_HMI.b1000_15_BuzzerResetPB,
    INT_PV := 0,
    BZ_OUT_BOOL => ARiBuzzerOut[2].11); // TIMER_ALARM
bInternalAlarm_b201_11_ThermalOilDownThermostatAlarm := arfbTimerAlarm[24].ALM_MSG_BOOL;

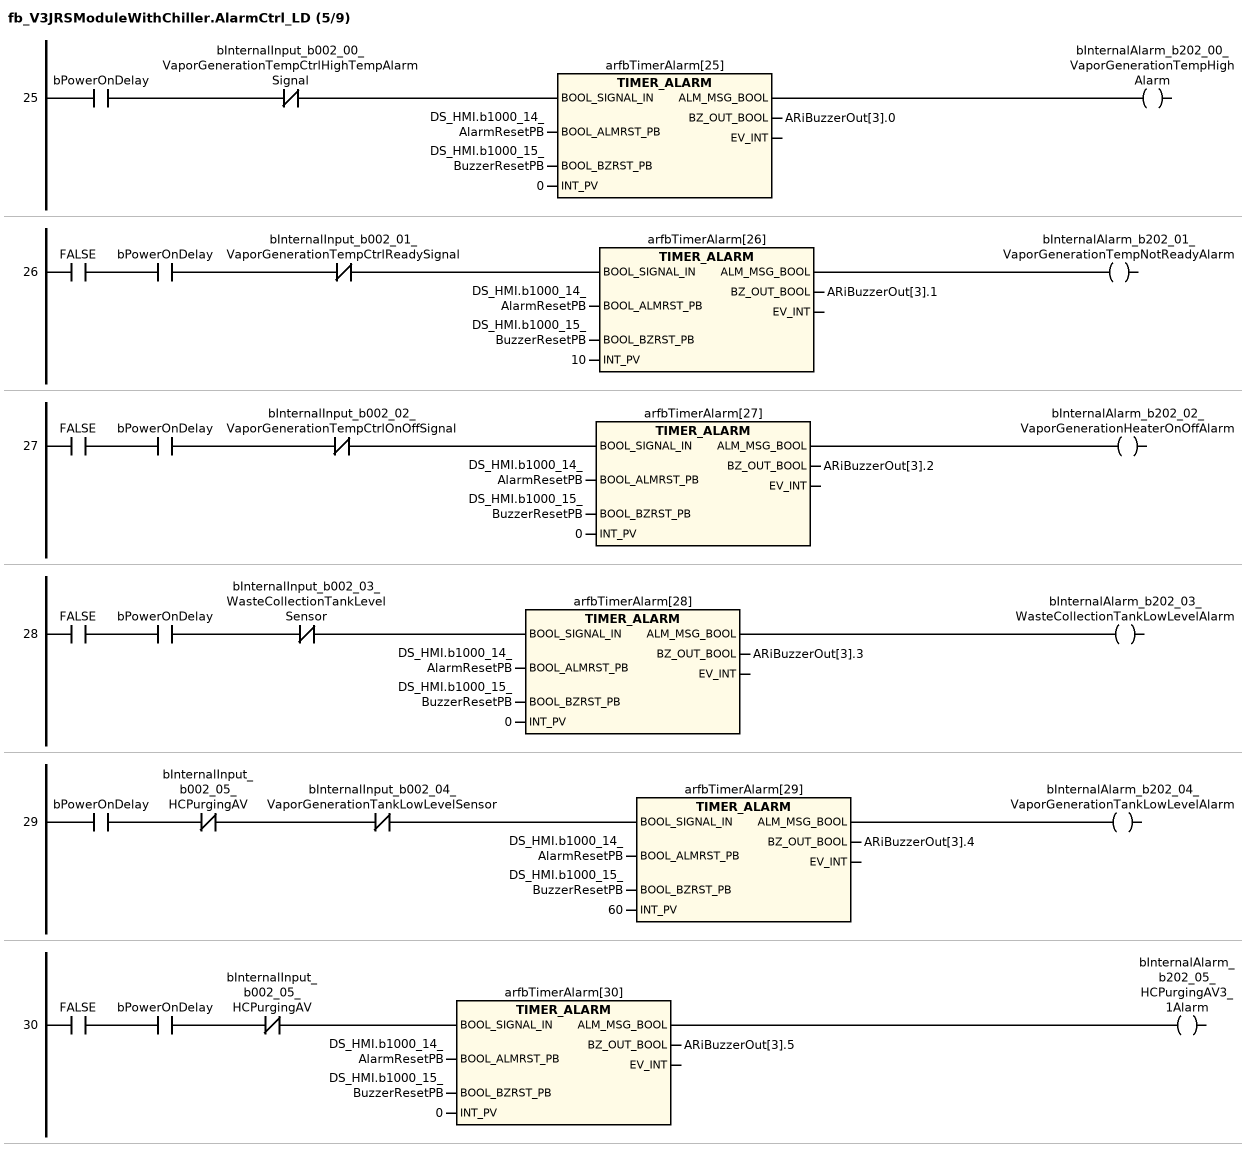
// NETWORK 25
arfbTimerAlarm[25](
    BOOL_SIGNAL_IN := bPowerOnDelay AND NOT bInternalInput_b002_00_VaporGenerationTempCtrlHighTempAlarmSignal,
    BOOL_ALMRST_PB := DS_HMI.b1000_14_AlarmResetPB,
    BOOL_BZRST_PB := DS_HMI.b1000_15_BuzzerResetPB,
    INT_PV := 0,
    BZ_OUT_BOOL => ARiBuzzerOut[3].0); // TIMER_ALARM
bInternalAlarm_b202_00_VaporGenerationTempHighAlarm := arfbTimerAlarm[25].ALM_MSG_BOOL;

// NETWORK 26
arfbTimerAlarm[26](
    BOOL_SIGNAL_IN := FALSE AND bPowerOnDelay AND NOT bInternalInput_b002_01_VaporGenerationTempCtrlReadySignal,
    BOOL_ALMRST_PB := DS_HMI.b1000_14_AlarmResetPB,
    BOOL_BZRST_PB := DS_HMI.b1000_15_BuzzerResetPB,
    INT_PV := 10,
    BZ_OUT_BOOL => ARiBuzzerOut[3].1); // TIMER_ALARM
bInternalAlarm_b202_01_VaporGenerationTempNotReadyAlarm := arfbTimerAlarm[26].ALM_MSG_BOOL;

// NETWORK 27
arfbTimerAlarm[27](
    BOOL_SIGNAL_IN := FALSE AND bPowerOnDelay AND NOT bInternalInput_b002_02_VaporGenerationTempCtrlOnOffSignal,
    BOOL_ALMRST_PB := DS_HMI.b1000_14_AlarmResetPB,
    BOOL_BZRST_PB := DS_HMI.b1000_15_BuzzerResetPB,
    INT_PV := 0,
    BZ_OUT_BOOL => ARiBuzzerOut[3].2); // TIMER_ALARM
bInternalAlarm_b202_02_VaporGenerationHeaterOnOffAlarm := arfbTimerAlarm[27].ALM_MSG_BOOL;

// NETWORK 28
arfbTimerAlarm[28](
    BOOL_SIGNAL_IN := FALSE AND bPowerOnDelay AND NOT bInternalInput_b002_03_WasteCollectionTankLevelSensor,
    BOOL_ALMRST_PB := DS_HMI.b1000_14_AlarmResetPB,
    BOOL_BZRST_PB := DS_HMI.b1000_15_BuzzerResetPB,
    INT_PV := 0,
    BZ_OUT_BOOL => ARiBuzzerOut[3].3); // TIMER_ALARM
bInternalAlarm_b202_03_WasteCollectionTankLowLevelAlarm := arfbTimerAlarm[28].ALM_MSG_BOOL;

// NETWORK 29
arfbTimerAlarm[29](
    BOOL_SIGNAL_IN := bPowerOnDelay AND NOT bInternalInput_b002_05_HCPurgingAV AND NOT bInternalInput_b002_04_VaporGenerationTankLowLevelSensor,
    BOOL_ALMRST_PB := DS_HMI.b1000_14_AlarmResetPB,
    BOOL_BZRST_PB := DS_HMI.b1000_15_BuzzerResetPB,
    INT_PV := 60,
    BZ_OUT_BOOL => ARiBuzzerOut[3].4); // TIMER_ALARM
bInternalAlarm_b202_04_VaporGenerationTankLowLevelAlarm := arfbTimerAlarm[29].ALM_MSG_BOOL;

// NETWORK 30
arfbTimerAlarm[30](
    BOOL_SIGNAL_IN := FALSE AND bPowerOnDelay AND NOT bInternalInput_b002_05_HCPurgingAV,
    BOOL_ALMRST_PB := DS_HMI.b1000_14_AlarmResetPB,
    BOOL_BZRST_PB := DS_HMI.b1000_15_BuzzerResetPB,
    INT_PV := 0,
    BZ_OUT_BOOL => ARiBuzzerOut[3].5); // TIMER_ALARM
bInternalAlarm_b202_05_HCPurgingAV3_1Alarm := arfbTimerAlarm[30].ALM_MSG_BOOL;

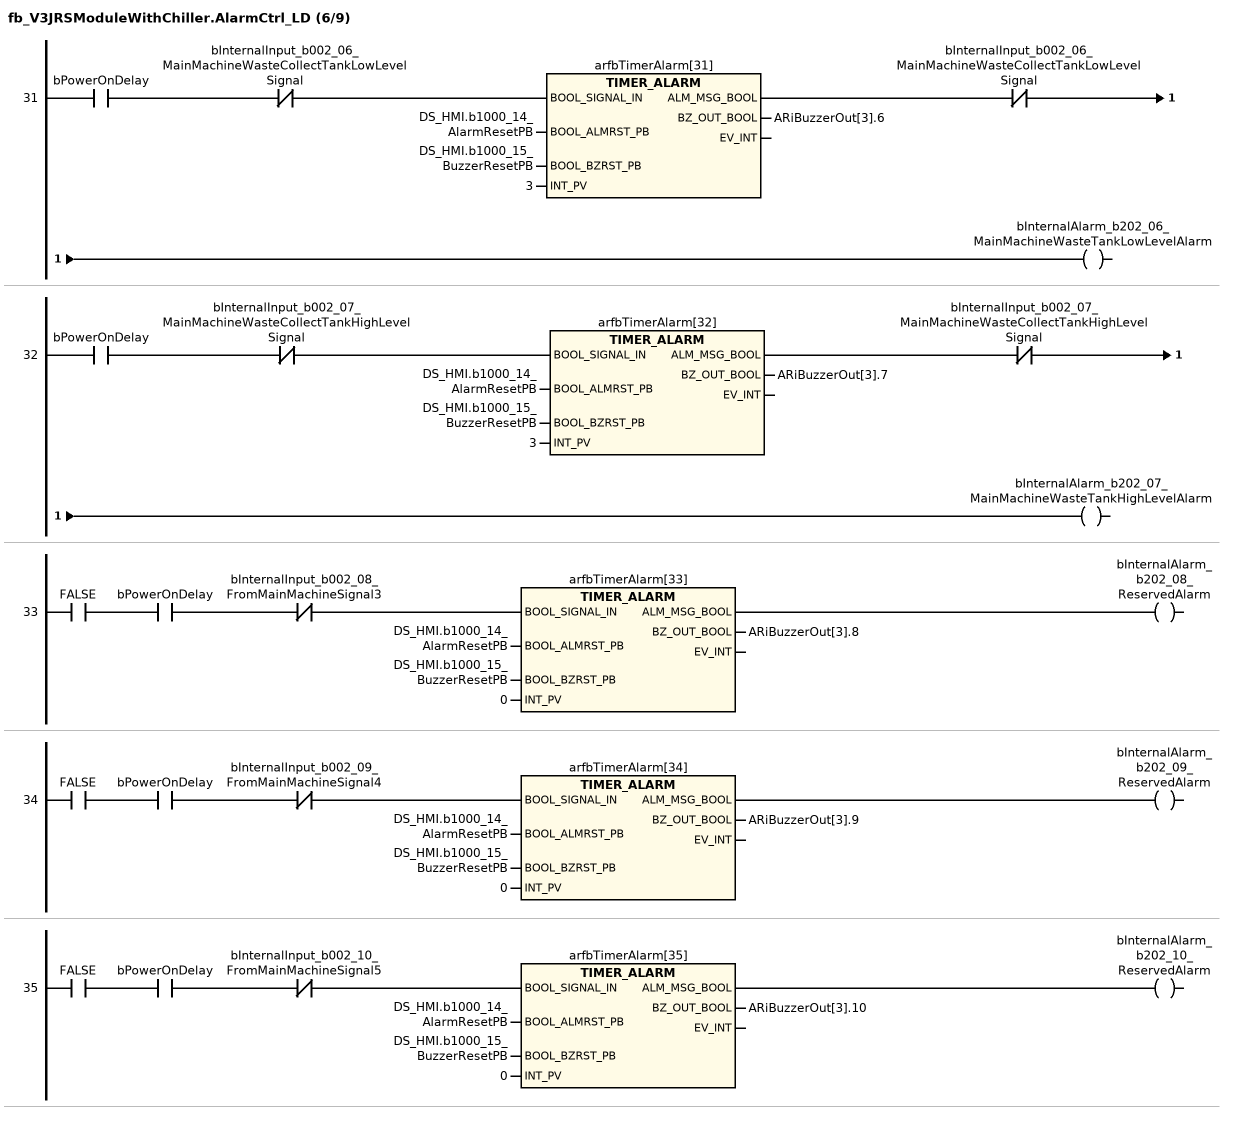
// NETWORK 31
arfbTimerAlarm[31](
    BOOL_SIGNAL_IN := bPowerOnDelay AND NOT bInternalInput_b002_06_MainMachineWasteCollectTankLowLevelSignal,
    BOOL_ALMRST_PB := DS_HMI.b1000_14_AlarmResetPB,
    BOOL_BZRST_PB := DS_HMI.b1000_15_BuzzerResetPB,
    INT_PV := 3,
    BZ_OUT_BOOL => ARiBuzzerOut[3].6); // TIMER_ALARM
bInternalAlarm_b202_06_MainMachineWasteTankLowLevelAlarm := arfbTimerAlarm[31].ALM_MSG_BOOL AND NOT bInternalInput_b002_06_MainMachineWasteCollectTankLowLevelSignal;

// NETWORK 32
arfbTimerAlarm[32](
    BOOL_SIGNAL_IN := bPowerOnDelay AND NOT bInternalInput_b002_07_MainMachineWasteCollectTankHighLevelSignal,
    BOOL_ALMRST_PB := DS_HMI.b1000_14_AlarmResetPB,
    BOOL_BZRST_PB := DS_HMI.b1000_15_BuzzerResetPB,
    INT_PV := 3,
    BZ_OUT_BOOL => ARiBuzzerOut[3].7); // TIMER_ALARM
bInternalAlarm_b202_07_MainMachineWasteTankHighLevelAlarm := arfbTimerAlarm[32].ALM_MSG_BOOL AND NOT bInternalInput_b002_07_MainMachineWasteCollectTankHighLevelSignal;

// NETWORK 33
arfbTimerAlarm[33](
    BOOL_SIGNAL_IN := FALSE AND bPowerOnDelay AND NOT bInternalInput_b002_08_FromMainMachineSignal3,
    BOOL_ALMRST_PB := DS_HMI.b1000_14_AlarmResetPB,
    BOOL_BZRST_PB := DS_HMI.b1000_15_BuzzerResetPB,
    INT_PV := 0,
    BZ_OUT_BOOL => ARiBuzzerOut[3].8); // TIMER_ALARM
bInternalAlarm_b202_08_ReservedAlarm := arfbTimerAlarm[33].ALM_MSG_BOOL;

// NETWORK 34
arfbTimerAlarm[34](
    BOOL_SIGNAL_IN := FALSE AND bPowerOnDelay AND NOT bInternalInput_b002_09_FromMainMachineSignal4,
    BOOL_ALMRST_PB := DS_HMI.b1000_14_AlarmResetPB,
    BOOL_BZRST_PB := DS_HMI.b1000_15_BuzzerResetPB,
    INT_PV := 0,
    BZ_OUT_BOOL => ARiBuzzerOut[3].9); // TIMER_ALARM
bInternalAlarm_b202_09_ReservedAlarm := arfbTimerAlarm[34].ALM_MSG_BOOL;

// NETWORK 35
arfbTimerAlarm[35](
    BOOL_SIGNAL_IN := FALSE AND bPowerOnDelay AND NOT bInternalInput_b002_10_FromMainMachineSignal5,
    BOOL_ALMRST_PB := DS_HMI.b1000_14_AlarmResetPB,
    BOOL_BZRST_PB := DS_HMI.b1000_15_BuzzerResetPB,
    INT_PV := 0,
    BZ_OUT_BOOL => ARiBuzzerOut[3].10); // TIMER_ALARM
bInternalAlarm_b202_10_ReservedAlarm := arfbTimerAlarm[35].ALM_MSG_BOOL;

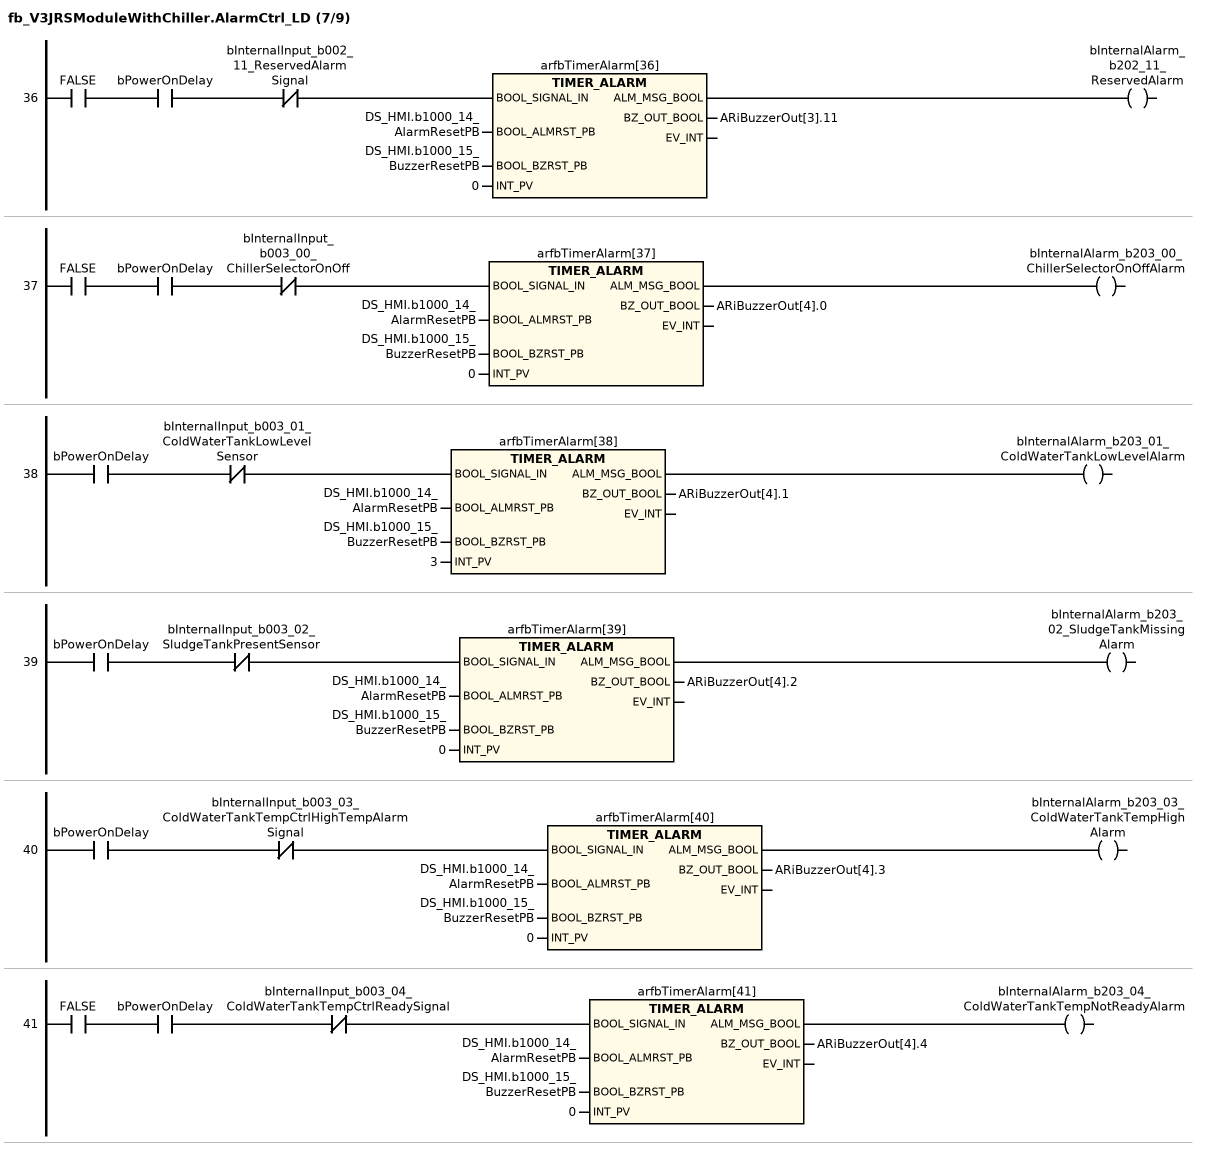
// NETWORK 36
arfbTimerAlarm[36](
    BOOL_SIGNAL_IN := FALSE AND bPowerOnDelay AND NOT bInternalInput_b002_11_ReservedAlarmSignal,
    BOOL_ALMRST_PB := DS_HMI.b1000_14_AlarmResetPB,
    BOOL_BZRST_PB := DS_HMI.b1000_15_BuzzerResetPB,
    INT_PV := 0,
    BZ_OUT_BOOL => ARiBuzzerOut[3].11); // TIMER_ALARM
bInternalAlarm_b202_11_ReservedAlarm := arfbTimerAlarm[36].ALM_MSG_BOOL;

// NETWORK 37
arfbTimerAlarm[37](
    BOOL_SIGNAL_IN := FALSE AND bPowerOnDelay AND NOT bInternalInput_b003_00_ChillerSelectorOnOff,
    BOOL_ALMRST_PB := DS_HMI.b1000_14_AlarmResetPB,
    BOOL_BZRST_PB := DS_HMI.b1000_15_BuzzerResetPB,
    INT_PV := 0,
    BZ_OUT_BOOL => ARiBuzzerOut[4].0); // TIMER_ALARM
bInternalAlarm_b203_00_ChillerSelectorOnOffAlarm := arfbTimerAlarm[37].ALM_MSG_BOOL;

// NETWORK 38
arfbTimerAlarm[38](
    BOOL_SIGNAL_IN := bPowerOnDelay AND NOT bInternalInput_b003_01_ColdWaterTankLowLevelSensor,
    BOOL_ALMRST_PB := DS_HMI.b1000_14_AlarmResetPB,
    BOOL_BZRST_PB := DS_HMI.b1000_15_BuzzerResetPB,
    INT_PV := 3,
    BZ_OUT_BOOL => ARiBuzzerOut[4].1); // TIMER_ALARM
bInternalAlarm_b203_01_ColdWaterTankLowLevelAlarm := arfbTimerAlarm[38].ALM_MSG_BOOL;

// NETWORK 39
arfbTimerAlarm[39](
    BOOL_SIGNAL_IN := bPowerOnDelay AND NOT bInternalInput_b003_02_SludgeTankPresentSensor,
    BOOL_ALMRST_PB := DS_HMI.b1000_14_AlarmResetPB,
    BOOL_BZRST_PB := DS_HMI.b1000_15_BuzzerResetPB,
    INT_PV := 0,
    BZ_OUT_BOOL => ARiBuzzerOut[4].2); // TIMER_ALARM
bInternalAlarm_b203_02_SludgeTankMissingAlarm := arfbTimerAlarm[39].ALM_MSG_BOOL;

// NETWORK 40
arfbTimerAlarm[40](
    BOOL_SIGNAL_IN := bPowerOnDelay AND NOT bInternalInput_b003_03_ColdWaterTankTempCtrlHighTempAlarmSignal,
    BOOL_ALMRST_PB := DS_HMI.b1000_14_AlarmResetPB,
    BOOL_BZRST_PB := DS_HMI.b1000_15_BuzzerResetPB,
    INT_PV := 0,
    BZ_OUT_BOOL => ARiBuzzerOut[4].3); // TIMER_ALARM
bInternalAlarm_b203_03_ColdWaterTankTempHighAlarm := arfbTimerAlarm[40].ALM_MSG_BOOL;

// NETWORK 41
arfbTimerAlarm[41](
    BOOL_SIGNAL_IN := FALSE AND bPowerOnDelay AND NOT bInternalInput_b003_04_ColdWaterTankTempCtrlReadySignal,
    BOOL_ALMRST_PB := DS_HMI.b1000_14_AlarmResetPB,
    BOOL_BZRST_PB := DS_HMI.b1000_15_BuzzerResetPB,
    INT_PV := 0,
    BZ_OUT_BOOL => ARiBuzzerOut[4].4); // TIMER_ALARM
bInternalAlarm_b203_04_ColdWaterTankTempNotReadyAlarm := arfbTimerAlarm[41].ALM_MSG_BOOL;

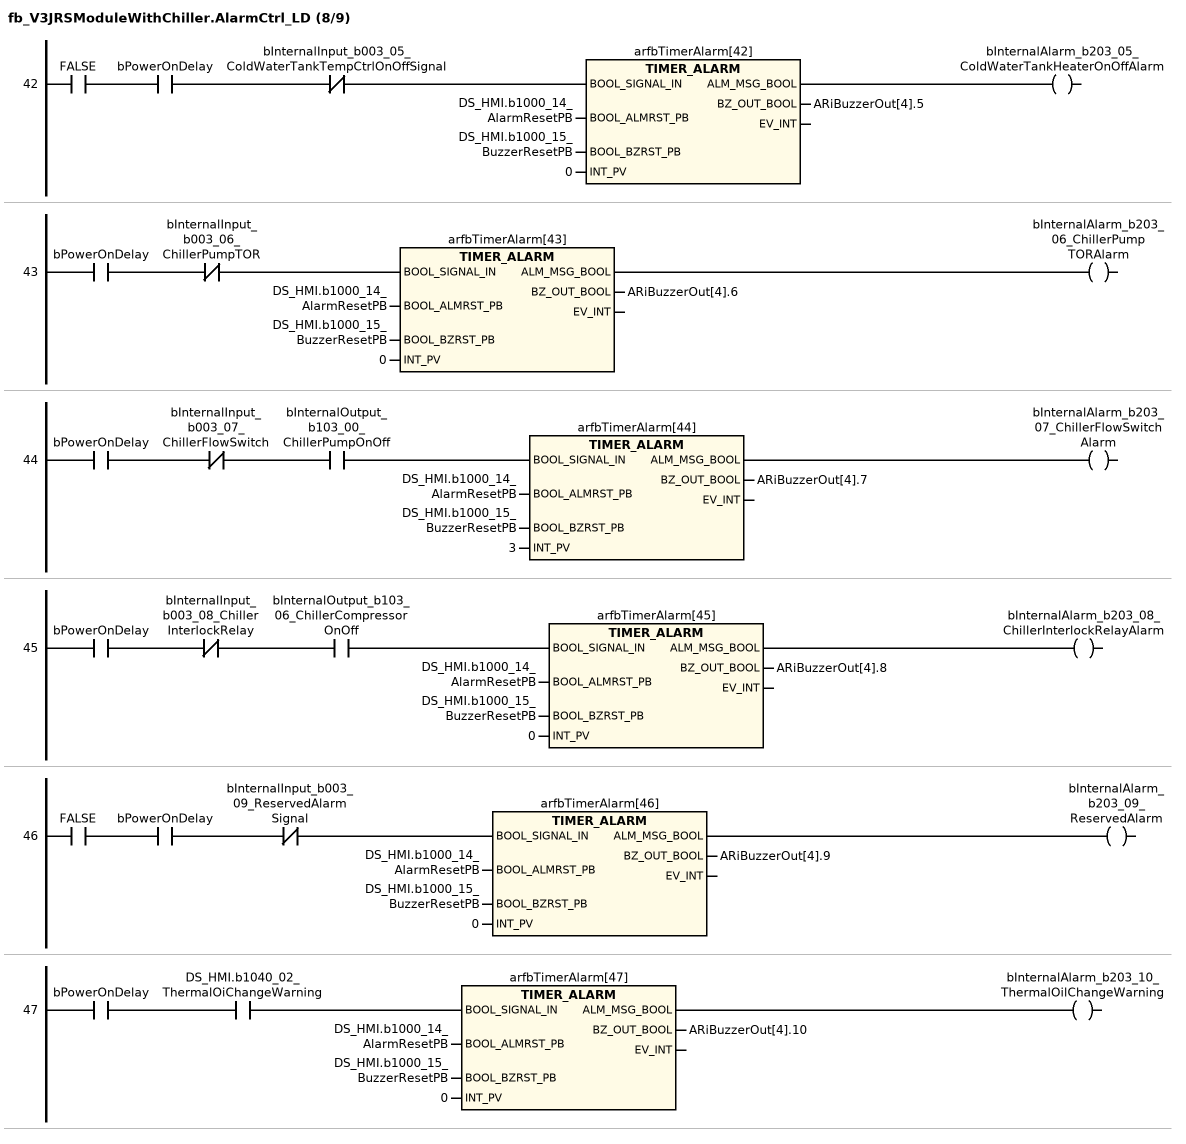
// NETWORK 42
arfbTimerAlarm[42](
    BOOL_SIGNAL_IN := FALSE AND bPowerOnDelay AND NOT bInternalInput_b003_05_ColdWaterTankTempCtrlOnOffSignal,
    BOOL_ALMRST_PB := DS_HMI.b1000_14_AlarmResetPB,
    BOOL_BZRST_PB := DS_HMI.b1000_15_BuzzerResetPB,
    INT_PV := 0,
    BZ_OUT_BOOL => ARiBuzzerOut[4].5); // TIMER_ALARM
bInternalAlarm_b203_05_ColdWaterTankHeaterOnOffAlarm := arfbTimerAlarm[42].ALM_MSG_BOOL;

// NETWORK 43
arfbTimerAlarm[43](
    BOOL_SIGNAL_IN := bPowerOnDelay AND NOT bInternalInput_b003_06_ChillerPumpTOR,
    BOOL_ALMRST_PB := DS_HMI.b1000_14_AlarmResetPB,
    BOOL_BZRST_PB := DS_HMI.b1000_15_BuzzerResetPB,
    INT_PV := 0,
    BZ_OUT_BOOL => ARiBuzzerOut[4].6); // TIMER_ALARM
bInternalAlarm_b203_06_ChillerPumpTORAlarm := arfbTimerAlarm[43].ALM_MSG_BOOL;

// NETWORK 44
arfbTimerAlarm[44](
    BOOL_SIGNAL_IN := bPowerOnDelay AND NOT bInternalInput_b003_07_ChillerFlowSwitch AND bInternalOutput_b103_00_ChillerPumpOnOff,
    BOOL_ALMRST_PB := DS_HMI.b1000_14_AlarmResetPB,
    BOOL_BZRST_PB := DS_HMI.b1000_15_BuzzerResetPB,
    INT_PV := 3,
    BZ_OUT_BOOL => ARiBuzzerOut[4].7); // TIMER_ALARM
bInternalAlarm_b203_07_ChillerFlowSwitchAlarm := arfbTimerAlarm[44].ALM_MSG_BOOL;

// NETWORK 45
arfbTimerAlarm[45](
    BOOL_SIGNAL_IN := bPowerOnDelay AND NOT bInternalInput_b003_08_ChillerInterlockRelay AND bInternalOutput_b103_06_ChillerCompressorOnOff,
    BOOL_ALMRST_PB := DS_HMI.b1000_14_AlarmResetPB,
    BOOL_BZRST_PB := DS_HMI.b1000_15_BuzzerResetPB,
    INT_PV := 0,
    BZ_OUT_BOOL => ARiBuzzerOut[4].8); // TIMER_ALARM
bInternalAlarm_b203_08_ChillerInterlockRelayAlarm := arfbTimerAlarm[45].ALM_MSG_BOOL;

// NETWORK 46
arfbTimerAlarm[46](
    BOOL_SIGNAL_IN := FALSE AND bPowerOnDelay AND NOT bInternalInput_b003_09_ReservedAlarmSignal,
    BOOL_ALMRST_PB := DS_HMI.b1000_14_AlarmResetPB,
    BOOL_BZRST_PB := DS_HMI.b1000_15_BuzzerResetPB,
    INT_PV := 0,
    BZ_OUT_BOOL => ARiBuzzerOut[4].9); // TIMER_ALARM
bInternalAlarm_b203_09_ReservedAlarm := arfbTimerAlarm[46].ALM_MSG_BOOL;

// NETWORK 47
arfbTimerAlarm[47](
    BOOL_SIGNAL_IN := bPowerOnDelay AND DS_HMI.b1040_02_ThermalOiChangeWarning,
    BOOL_ALMRST_PB := DS_HMI.b1000_14_AlarmResetPB,
    BOOL_BZRST_PB := DS_HMI.b1000_15_BuzzerResetPB,
    INT_PV := 0,
    BZ_OUT_BOOL => ARiBuzzerOut[4].10); // TIMER_ALARM
bInternalAlarm_b203_10_ThermalOilChangeWarning := arfbTimerAlarm[47].ALM_MSG_BOOL;

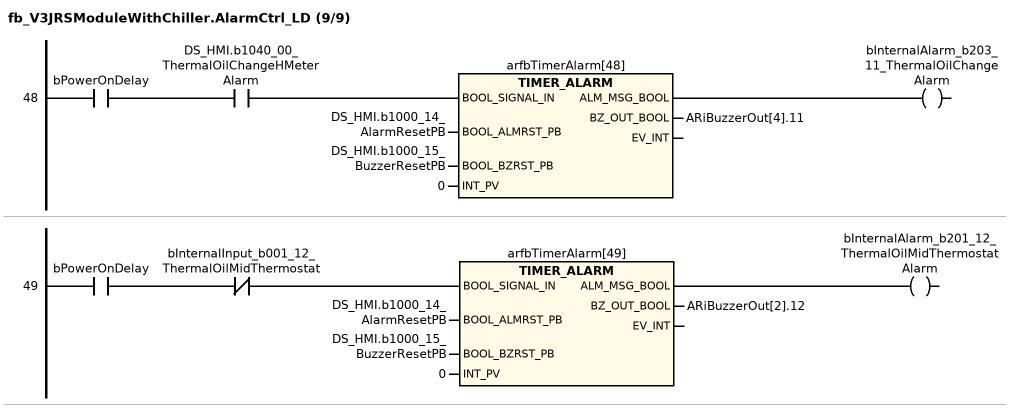
// NETWORK 48
arfbTimerAlarm[48](
    BOOL_SIGNAL_IN := bPowerOnDelay AND DS_HMI.b1040_00_ThermalOilChangeHMeterAlarm,
    BOOL_ALMRST_PB := DS_HMI.b1000_14_AlarmResetPB,
    BOOL_BZRST_PB := DS_HMI.b1000_15_BuzzerResetPB,
    INT_PV := 0,
    BZ_OUT_BOOL => ARiBuzzerOut[4].11); // TIMER_ALARM
bInternalAlarm_b203_11_ThermalOilChangeAlarm := arfbTimerAlarm[48].ALM_MSG_BOOL;

// NETWORK 49
arfbTimerAlarm[49](
    BOOL_SIGNAL_IN := bPowerOnDelay AND NOT bInternalInput_b001_12_ThermalOilMidThermostat,
    BOOL_ALMRST_PB := DS_HMI.b1000_14_AlarmResetPB,
    BOOL_BZRST_PB := DS_HMI.b1000_15_BuzzerResetPB,
    INT_PV := 0,
    BZ_OUT_BOOL => ARiBuzzerOut[2].12); // TIMER_ALARM
bInternalAlarm_b201_12_ThermalOilMidThermostatAlarm := arfbTimerAlarm[49].ALM_MSG_BOOL;
END_ACTION

ACTION AutoBoilingCtrl_LD:
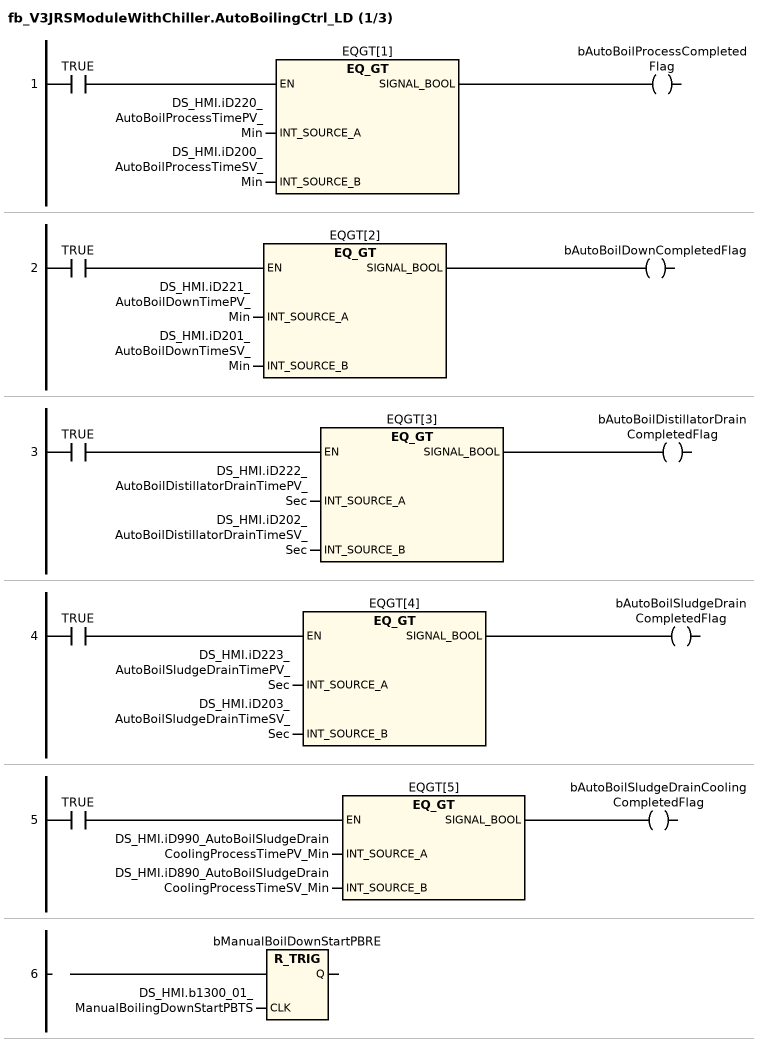
// NETWORK 1
EQGT[1](INT_SOURCE_A := DS_HMI.iD220_AutoBoilProcessTimePV_Min, INT_SOURCE_B := DS_HMI.iD200_AutoBoilProcessTimeSV_Min); // EQ_GT
bAutoBoilProcessCompletedFlag := EQGT[1].SIGNAL_BOOL;

// NETWORK 2
EQGT[2](INT_SOURCE_A := DS_HMI.iD221_AutoBoilDownTimePV_Min, INT_SOURCE_B := DS_HMI.iD201_AutoBoilDownTimeSV_Min); // EQ_GT
bAutoBoilDownCompletedFlag := EQGT[2].SIGNAL_BOOL;

// NETWORK 3
EQGT[3](INT_SOURCE_A := DS_HMI.iD222_AutoBoilDistillatorDrainTimePV_Sec, INT_SOURCE_B := DS_HMI.iD202_AutoBoilDistillatorDrainTimeSV_Sec); // EQ_GT
bAutoBoilDistillatorDrainCompletedFlag := EQGT[3].SIGNAL_BOOL;

// NETWORK 4
EQGT[4](INT_SOURCE_A := DS_HMI.iD223_AutoBoilSludgeDrainTimePV_Sec, INT_SOURCE_B := DS_HMI.iD203_AutoBoilSludgeDrainTimeSV_Sec); // EQ_GT
bAutoBoilSludgeDrainCompletedFlag := EQGT[4].SIGNAL_BOOL;

// NETWORK 5
EQGT[5](INT_SOURCE_A := DS_HMI.iD990_AutoBoilSludgeDrainCoolingProcessTimePV_Min, INT_SOURCE_B := DS_HMI.iD890_AutoBoilSludgeDrainCoolingProcessTimeSV_Min); // EQ_GT
bAutoBoilSludgeDrainCoolingCompletedFlag := EQGT[5].SIGNAL_BOOL;

// NETWORK 6
bManualBoilDownStartPBRE(CLK := DS_HMI.b1300_01_ManualBoilingDownStartPBTS); // R_TRIG

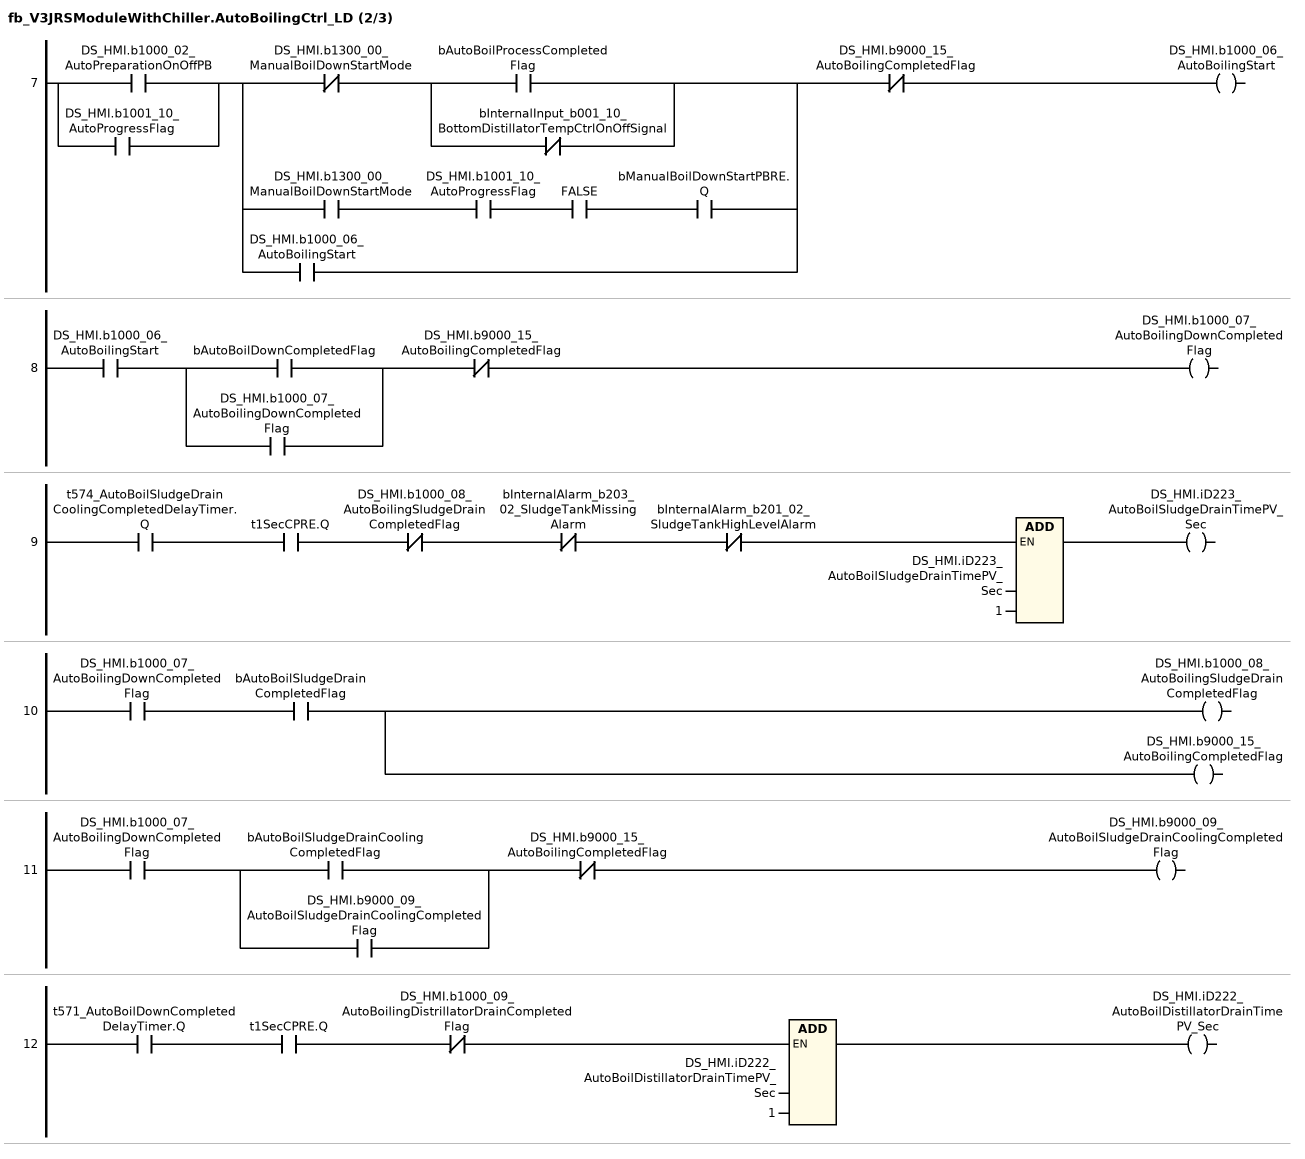
// NETWORK 7
DS_HMI.b1000_06_AutoBoilingStart := ((DS_HMI.b1000_02_AutoPreparationOnOffPB OR DS_HMI.b1001_10_AutoProgressFlag) AND (NOT DS_HMI.b1300_00_ManualBoilDownStartMode AND (bAutoBoilProcessCompletedFlag OR NOT bInternalInput_b001_10_BottomDistillatorTempCtrlOnOffSignal) OR DS_HMI.b1300_00_ManualBoilDownStartMode AND DS_HMI.b1001_10_AutoProgressFlag AND FALSE AND bManualBoilDownStartPBRE.Q OR DS_HMI.b1000_06_AutoBoilingStart)) AND NOT DS_HMI.b9000_15_AutoBoilingCompletedFlag;

// NETWORK 8
DS_HMI.b1000_07_AutoBoilingDownCompletedFlag := (DS_HMI.b1000_06_AutoBoilingStart AND (bAutoBoilDownCompletedFlag OR DS_HMI.b1000_07_AutoBoilingDownCompletedFlag)) AND NOT DS_HMI.b9000_15_AutoBoilingCompletedFlag;

// NETWORK 9
IF t574_AutoBoilSludgeDrainCoolingCompletedDelayTimer.Q AND t1SecCPRE.Q AND NOT DS_HMI.b1000_08_AutoBoilingSludgeDrainCompletedFlag AND NOT bInternalAlarm_b203_02_SludgeTankMissingAlarm AND NOT bInternalAlarm_b201_02_SludgeTankHighLevelAlarm THEN
    _w1 := DS_HMI.iD223_AutoBoilSludgeDrainTimePV_Sec + 1;
END_IF
DS_HMI.iD223_AutoBoilSludgeDrainTimePV_Sec := _w1;

// NETWORK 10
_w2 := DS_HMI.b1000_07_AutoBoilingDownCompletedFlag AND bAutoBoilSludgeDrainCompletedFlag;
DS_HMI.b1000_08_AutoBoilingSludgeDrainCompletedFlag := _w2;
DS_HMI.b9000_15_AutoBoilingCompletedFlag := _w2;

// NETWORK 11
DS_HMI.b9000_09_AutoBoilSludgeDrainCoolingCompletedFlag := (DS_HMI.b1000_07_AutoBoilingDownCompletedFlag AND (bAutoBoilSludgeDrainCoolingCompletedFlag OR DS_HMI.b9000_09_AutoBoilSludgeDrainCoolingCompletedFlag)) AND NOT DS_HMI.b9000_15_AutoBoilingCompletedFlag;

// NETWORK 12
IF t571_AutoBoilDownCompletedDelayTimer.Q AND t1SecCPRE.Q AND NOT DS_HMI.b1000_09_AutoBoilingDistrillatorDrainCompletedFlag THEN
    _w3 := DS_HMI.iD222_AutoBoilDistillatorDrainTimePV_Sec + 1;
END_IF
DS_HMI.iD222_AutoBoilDistillatorDrainTimePV_Sec := _w3;

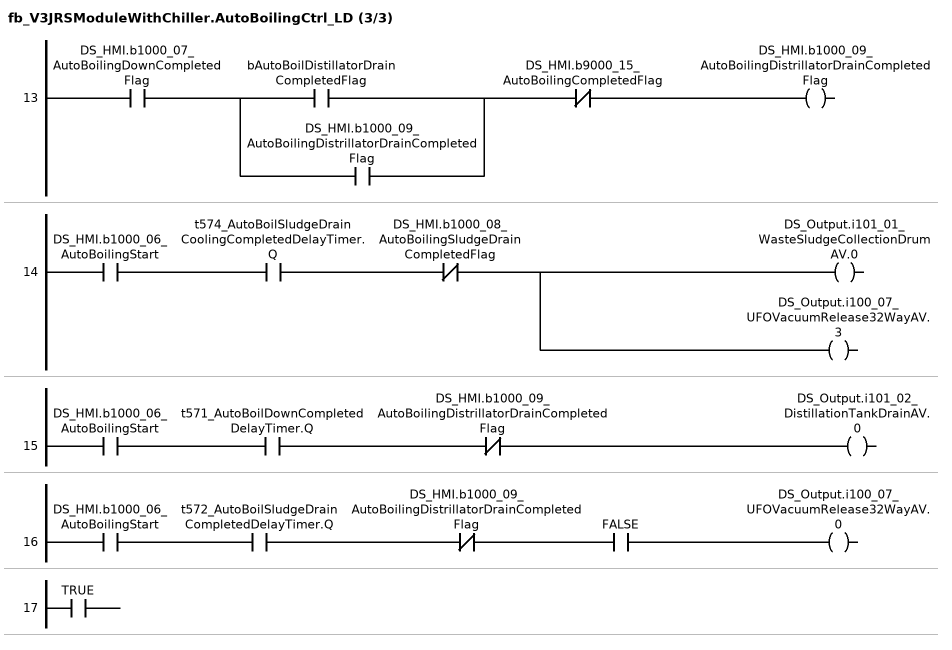
// NETWORK 13
DS_HMI.b1000_09_AutoBoilingDistrillatorDrainCompletedFlag := (DS_HMI.b1000_07_AutoBoilingDownCompletedFlag AND (bAutoBoilDistillatorDrainCompletedFlag OR DS_HMI.b1000_09_AutoBoilingDistrillatorDrainCompletedFlag)) AND NOT DS_HMI.b9000_15_AutoBoilingCompletedFlag;

// NETWORK 14
_w4 := DS_HMI.b1000_06_AutoBoilingStart AND t574_AutoBoilSludgeDrainCoolingCompletedDelayTimer.Q AND NOT DS_HMI.b1000_08_AutoBoilingSludgeDrainCompletedFlag;
DS_Output.i101_01_WasteSludgeCollectionDrumAV.0 := _w4;
DS_Output.i100_07_UFOVacuumRelease32WayAV.3 := _w4;

// NETWORK 15
DS_Output.i101_02_DistillationTankDrainAV.0 := DS_HMI.b1000_06_AutoBoilingStart AND t571_AutoBoilDownCompletedDelayTimer.Q AND NOT DS_HMI.b1000_09_AutoBoilingDistrillatorDrainCompletedFlag;

// NETWORK 16
DS_Output.i100_07_UFOVacuumRelease32WayAV.0 := DS_HMI.b1000_06_AutoBoilingStart AND t572_AutoBoilSludgeDrainCompletedDelayTimer.Q AND NOT DS_HMI.b1000_09_AutoBoilingDistrillatorDrainCompletedFlag AND FALSE;

// NETWORK 17
END_ACTION

ACTION AutoBoilingCtrl_ST:
	(*Timer*)
	t570_AutoBoilingStartDelayTimer(IN:=DS_HMI.b1000_06_AutoBoilingStart , PT:=t#1s , Q=> , ET=> );
	t571_AutoBoilDownCompletedDelayTimer(IN:=DS_HMI.b1000_07_AutoBoilingDownCompletedFlag , PT:=t#1s , Q=> , ET=> );
	t572_AutoBoilSludgeDrainCompletedDelayTimer(IN:=DS_HMI.b1000_08_AutoBoilingSludgeDrainCompletedFlag , PT:=t#1s , Q=> , ET=> );
	t573_AutoBoilDistillatorDrainCompletedDelayTimer(IN:=DS_HMI.b1000_09_AutoBoilingDistrillatorDrainCompletedFlag , PT:=t#1s , Q=> , ET=> );

	t574_AutoBoilSludgeDrainCoolingCompletedDelayTimer(IN:=DS_HMI.b9000_09_AutoBoilSludgeDrainCoolingCompletedFlag , PT:=t#1s , Q=> , ET=> );  (************* New extra request by customer - YCH************)


	(*AutoBoiling Boil Process Time Counting*)
	IF DS_HMI.b1001_10_AutoProgressFlag
	AND NOT DS_HMI.b1300_00_ManualBoilDownStartMode
	AND t1SecCPRE.Q
	THEN

		IF NOT DS_HMI.b1000_06_AutoBoilingStart THEN

			DS_HMI.iD225_AutoBoilProcessTimePV_Sec := DS_HMI.iD225_AutoBoilProcessTimePV_Sec + 1;

			IF DS_HMI.iD225_AutoBoilProcessTimePV_Sec > 59 THEN
				DS_HMI.iD220_AutoBoilProcessTimePV_Min := DS_HMI.iD220_AutoBoilProcessTimePV_Min + 1;
				DS_HMI.iD225_AutoBoilProcessTimePV_Sec := 0;
			END_IF

		END_IF

	END_IF

	(*AutoBoiling Boil Down Time Counting*)

	IF t570_AutoBoilingStartDelayTimer.Q
	AND t1SecCPRE.Q
	THEN

		IF NOT DS_HMI.b1000_07_AutoBoilingDownCompletedFlag THEN

			DS_HMI.iD226_AutoBoilDownTimePV_Sec := DS_HMI.iD226_AutoBoilDownTimePV_Sec + 1;

			IF DS_HMI.iD226_AutoBoilDownTimePV_Sec > 59 THEN
				DS_HMI.iD221_AutoBoilDownTimePV_Min := DS_HMI.iD221_AutoBoilDownTimePV_Min + 1;
				DS_HMI.iD226_AutoBoilDownTimePV_Sec := 0;
			END_IF

		END_IF

	END_IF


	(*AutoBoiling Sludge Drain Cooling Time Counting*)       (************* New extra request by customer - YCH************)

	IF t573_AutoBoilDistillatorDrainCompletedDelayTimer.Q
	AND t1SecCPRE.Q
	THEN

		IF NOT DS_HMI.b9000_09_AutoBoilSludgeDrainCoolingCompletedFlag THEN

			DS_HMI.iD991_AutoBoilSludgeDrainCoolingProcessTimePV_Sec := DS_HMI.iD991_AutoBoilSludgeDrainCoolingProcessTimePV_Sec + 1;

			IF DS_HMI.iD991_AutoBoilSludgeDrainCoolingProcessTimePV_Sec > 59 THEN
				DS_HMI.iD990_AutoBoilSludgeDrainCoolingProcessTimePV_Min := DS_HMI.iD990_AutoBoilSludgeDrainCoolingProcessTimePV_Min + 1;
				DS_HMI.iD991_AutoBoilSludgeDrainCoolingProcessTimePV_Sec := 0;
			END_IF

		END_IF

	END_IF


	(*Auto Boiling Reset*)
	IF DS_HMI.b9000_15_AutoBoilingCompletedFlag OR  t592_ManualBoilSludgeDrainCompletedDelayTimer.Q (*t572_AutoBoilSludgeDrainCompletedDelayTimer.Q*) THEN
	
		DS_HMI.iD220_AutoBoilProcessTimePV_Min						:= 0;
		DS_HMI.iD221_AutoBoilDownTimePV_Min						:= 0;
		DS_HMI.iD990_AutoBoilSludgeDrainCoolingProcessTimePV_Min 	:= 0; (************* New extra request by customer - YCH************)
		DS_HMI.iD222_AutoBoilDistillatorDrainTimePV_Sec				:= 0;
		DS_HMI.iD223_AutoBoilSludgeDrainTimePV_Sec					:= 0;
		DS_HMI.iD225_AutoBoilProcessTimePV_Sec						:= 0;
		DS_HMI.iD226_AutoBoilDownTimePV_Sec						:= 0;
		DS_HMI.iD991_AutoBoilSludgeDrainCoolingProcessTimePV_Sec 	:= 0; (************* New extra request by customer - YCH************)

		DS_HMI.b1300_01_ManualBoilingDownStartPBTS 			:= FALSE;

	END_IF

	IF NOT DS_HMI.b1300_00_ManualBoilDownStartMode THEN
		DS_HMI.b1300_01_ManualBoilingDownStartPBTS 			:= FALSE;
	END_IF
END_ACTION

ACTION AutoCtrl_LD:
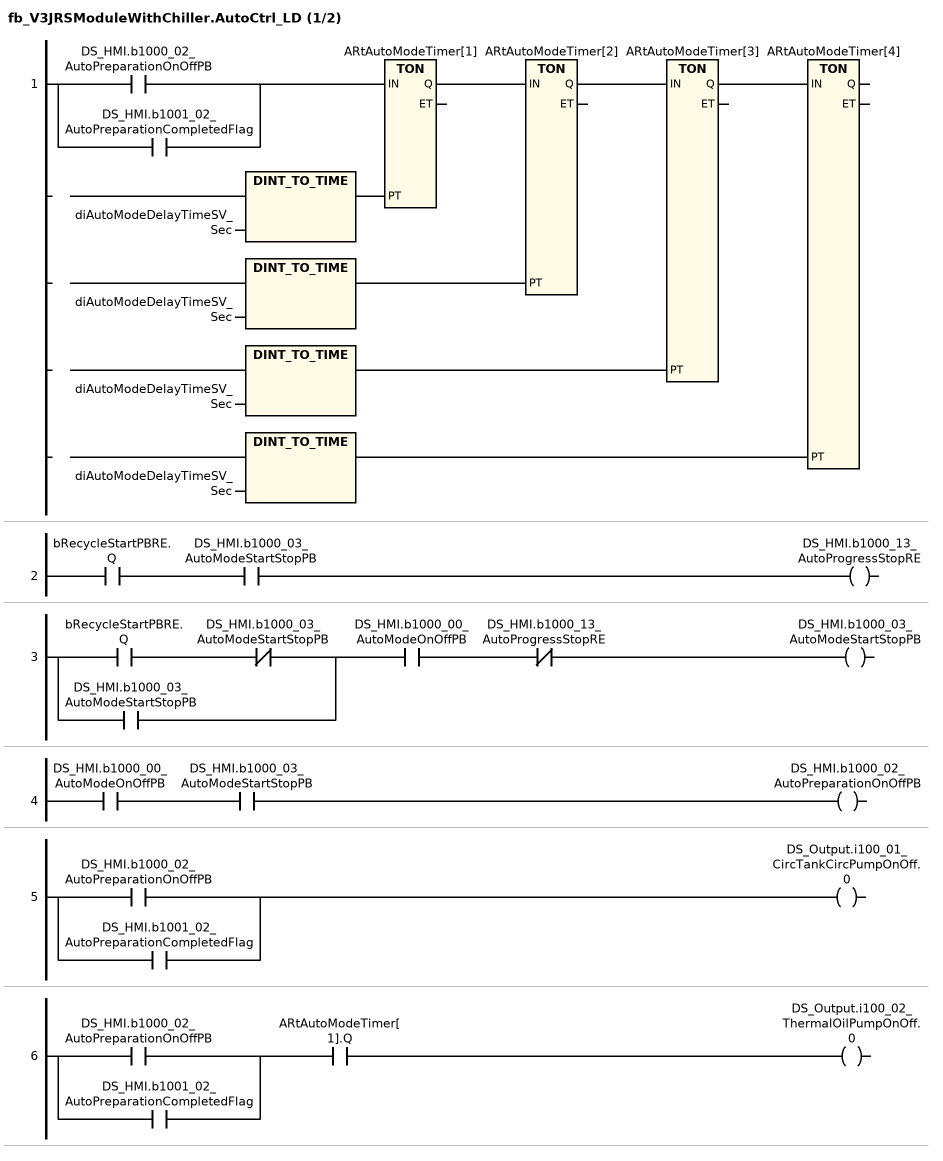
// NETWORK 1
ARtAutoModeTimer[1](IN := DS_HMI.b1000_02_AutoPreparationOnOffPB OR DS_HMI.b1001_02_AutoPreparationCompletedFlag, PT := DINT_TO_TIME(diAutoModeDelayTimeSV_Sec)); // TON
ARtAutoModeTimer[2](IN := ARtAutoModeTimer[1].Q, PT := DINT_TO_TIME(diAutoModeDelayTimeSV_Sec)); // TON
ARtAutoModeTimer[3](IN := ARtAutoModeTimer[2].Q, PT := DINT_TO_TIME(diAutoModeDelayTimeSV_Sec)); // TON
ARtAutoModeTimer[4](IN := ARtAutoModeTimer[3].Q, PT := DINT_TO_TIME(diAutoModeDelayTimeSV_Sec)); // TON

// NETWORK 2
DS_HMI.b1000_13_AutoProgressStopRE := bRecycleStartPBRE.Q AND DS_HMI.b1000_03_AutoModeStartStopPB;

// NETWORK 3
DS_HMI.b1000_03_AutoModeStartStopPB := (bRecycleStartPBRE.Q AND NOT DS_HMI.b1000_03_AutoModeStartStopPB OR DS_HMI.b1000_03_AutoModeStartStopPB) AND DS_HMI.b1000_00_AutoModeOnOffPB AND NOT DS_HMI.b1000_13_AutoProgressStopRE;

// NETWORK 4
DS_HMI.b1000_02_AutoPreparationOnOffPB := DS_HMI.b1000_00_AutoModeOnOffPB AND DS_HMI.b1000_03_AutoModeStartStopPB;

// NETWORK 5
DS_Output.i100_01_CircTankCircPumpOnOff.0 := DS_HMI.b1000_02_AutoPreparationOnOffPB OR DS_HMI.b1001_02_AutoPreparationCompletedFlag;

// NETWORK 6
DS_Output.i100_02_ThermalOilPumpOnOff.0 := (DS_HMI.b1000_02_AutoPreparationOnOffPB OR DS_HMI.b1001_02_AutoPreparationCompletedFlag) AND ARtAutoModeTimer[1].Q;

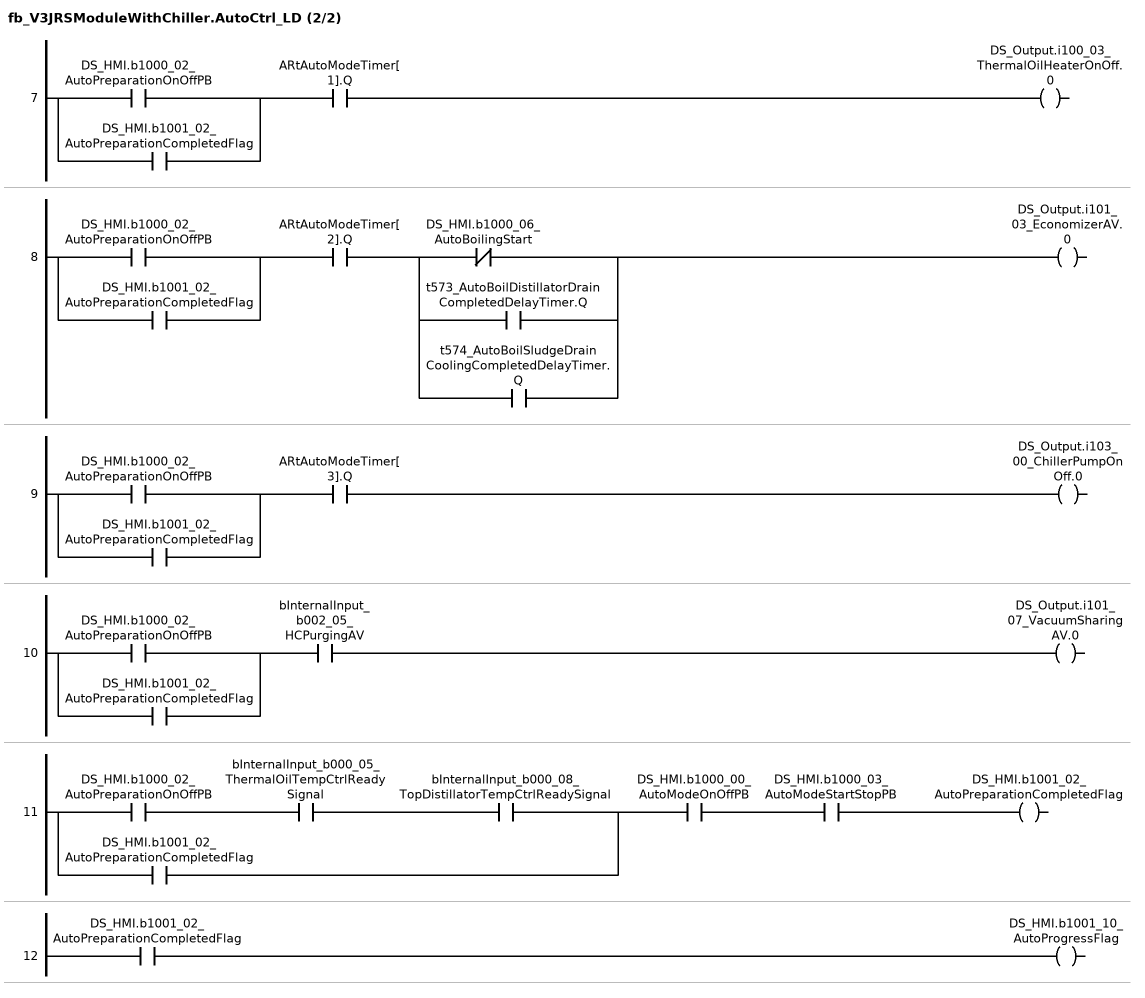
// NETWORK 7
DS_Output.i100_03_ThermalOilHeaterOnOff.0 := (DS_HMI.b1000_02_AutoPreparationOnOffPB OR DS_HMI.b1001_02_AutoPreparationCompletedFlag) AND ARtAutoModeTimer[1].Q;

// NETWORK 8
DS_Output.i101_03_EconomizerAV.0 := (DS_HMI.b1000_02_AutoPreparationOnOffPB OR DS_HMI.b1001_02_AutoPreparationCompletedFlag) AND ARtAutoModeTimer[2].Q AND (NOT DS_HMI.b1000_06_AutoBoilingStart OR t573_AutoBoilDistillatorDrainCompletedDelayTimer.Q OR t574_AutoBoilSludgeDrainCoolingCompletedDelayTimer.Q);

// NETWORK 9
DS_Output.i103_00_ChillerPumpOnOff.0 := (DS_HMI.b1000_02_AutoPreparationOnOffPB OR DS_HMI.b1001_02_AutoPreparationCompletedFlag) AND ARtAutoModeTimer[3].Q;

// NETWORK 10
DS_Output.i101_07_VacuumSharingAV.0 := (DS_HMI.b1000_02_AutoPreparationOnOffPB OR DS_HMI.b1001_02_AutoPreparationCompletedFlag) AND bInternalInput_b002_05_HCPurgingAV;

// NETWORK 11
DS_HMI.b1001_02_AutoPreparationCompletedFlag := (DS_HMI.b1000_02_AutoPreparationOnOffPB AND bInternalInput_b000_05_ThermalOilTempCtrlReadySignal AND bInternalInput_b000_08_TopDistillatorTempCtrlReadySignal OR DS_HMI.b1001_02_AutoPreparationCompletedFlag) AND DS_HMI.b1000_00_AutoModeOnOffPB AND DS_HMI.b1000_03_AutoModeStartStopPB;

// NETWORK 12
DS_HMI.b1001_10_AutoProgressFlag := DS_HMI.b1001_02_AutoPreparationCompletedFlag;
END_ACTION

ACTION AutoHCTopUp_LD:
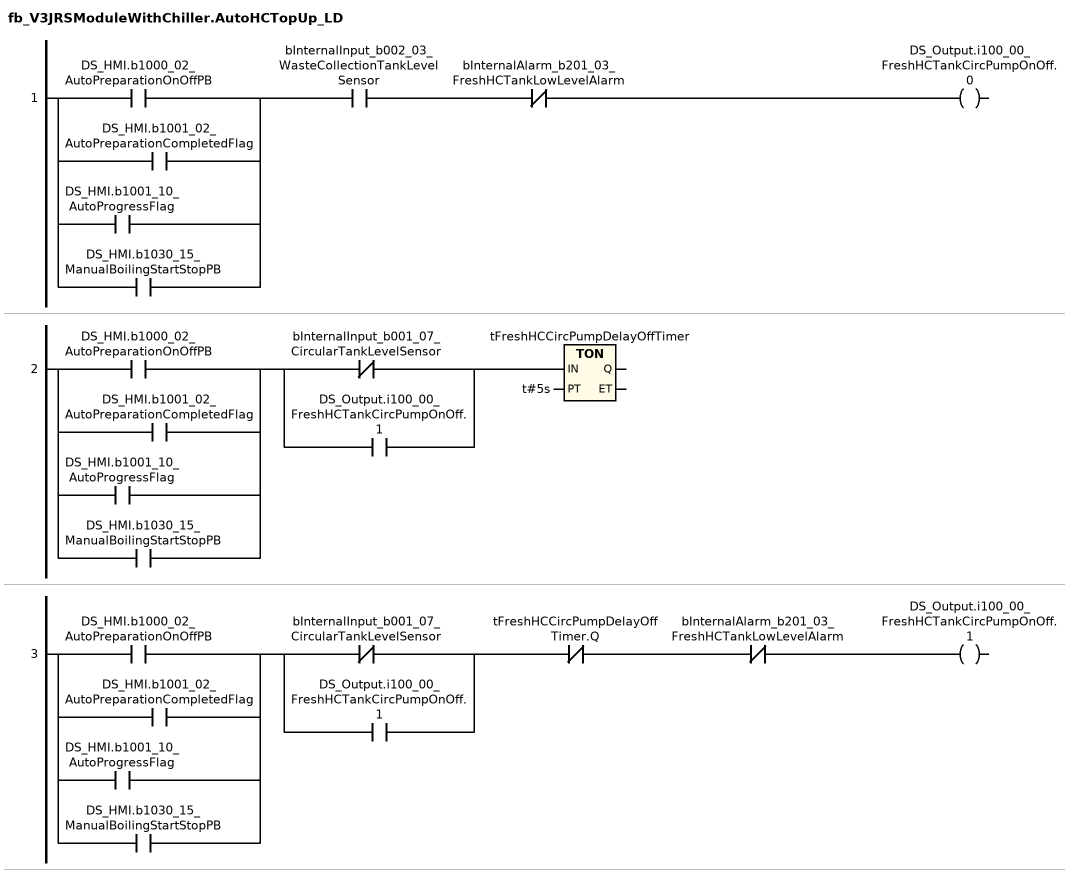
// NETWORK 1
DS_Output.i100_00_FreshHCTankCircPumpOnOff.0 := (DS_HMI.b1000_02_AutoPreparationOnOffPB OR DS_HMI.b1001_02_AutoPreparationCompletedFlag OR DS_HMI.b1001_10_AutoProgressFlag OR DS_HMI.b1030_15_ManualBoilingStartStopPB) AND bInternalInput_b002_03_WasteCollectionTankLevelSensor AND NOT bInternalAlarm_b201_03_FreshHCTankLowLevelAlarm;

// NETWORK 2
tFreshHCCircPumpDelayOffTimer(IN := (DS_HMI.b1000_02_AutoPreparationOnOffPB OR DS_HMI.b1001_02_AutoPreparationCompletedFlag OR DS_HMI.b1001_10_AutoProgressFlag OR DS_HMI.b1030_15_ManualBoilingStartStopPB) AND (NOT bInternalInput_b001_07_CircularTankLevelSensor OR DS_Output.i100_00_FreshHCTankCircPumpOnOff.1), PT := t#5s); // TON

// NETWORK 3
DS_Output.i100_00_FreshHCTankCircPumpOnOff.1 := ((DS_HMI.b1000_02_AutoPreparationOnOffPB OR DS_HMI.b1001_02_AutoPreparationCompletedFlag OR DS_HMI.b1001_10_AutoProgressFlag OR DS_HMI.b1030_15_ManualBoilingStartStopPB) AND (NOT bInternalInput_b001_07_CircularTankLevelSensor OR DS_Output.i100_00_FreshHCTankCircPumpOnOff.1)) AND NOT tFreshHCCircPumpDelayOffTimer.Q AND NOT bInternalAlarm_b201_03_FreshHCTankLowLevelAlarm;
END_ACTION

ACTION BuzzerCtrl_ST:
IF ARiBuzzerOut[1] <>0
AND ARiBuzzerOut[2] <> 0
AND ARiBuzzerOut[3] <> 0
AND ARiBuzzerOut[4] <> 0
THEN
DS_Output.i100_04_Buzzer.0 := TRUE;
ELSE
DS_Output.i100_04_Buzzer.0 := FALSE;
END_IF
END_ACTION

ACTION ChillerCtrl_LD:
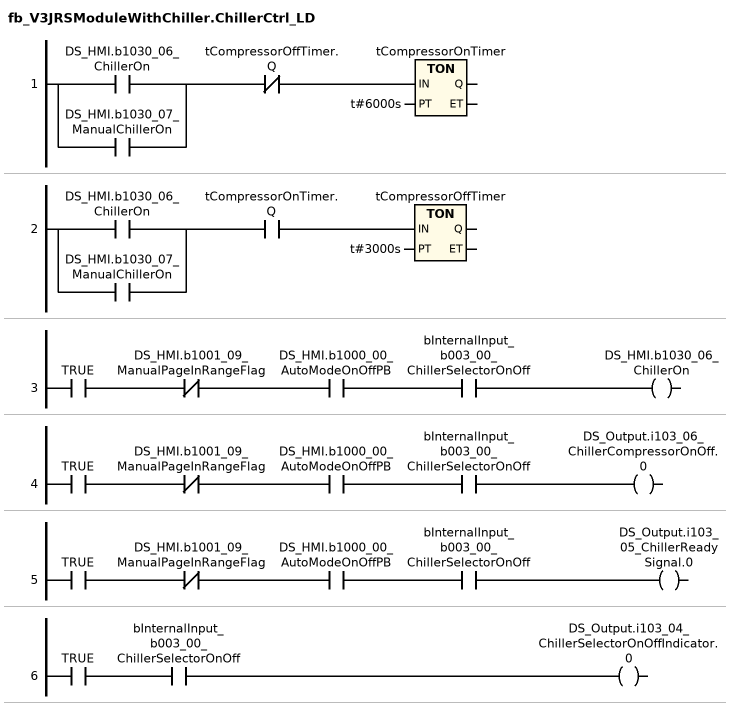
// NETWORK 1
tCompressorOnTimer(IN := (DS_HMI.b1030_06_ChillerOn OR DS_HMI.b1030_07_ManualChillerOn) AND NOT tCompressorOffTimer.Q, PT := t#6000s); // TON

// NETWORK 2
tCompressorOffTimer(IN := (DS_HMI.b1030_06_ChillerOn OR DS_HMI.b1030_07_ManualChillerOn) AND tCompressorOnTimer.Q, PT := t#3000s); // TON

// NETWORK 3
DS_HMI.b1030_06_ChillerOn := TRUE AND NOT DS_HMI.b1001_09_ManualPageInRangeFlag AND DS_HMI.b1000_00_AutoModeOnOffPB AND bInternalInput_b003_00_ChillerSelectorOnOff;

// NETWORK 4
DS_Output.i103_06_ChillerCompressorOnOff.0 := TRUE AND NOT DS_HMI.b1001_09_ManualPageInRangeFlag AND DS_HMI.b1000_00_AutoModeOnOffPB AND bInternalInput_b003_00_ChillerSelectorOnOff;

// NETWORK 5
DS_Output.i103_05_ChillerReadySignal.0 := TRUE AND NOT DS_HMI.b1001_09_ManualPageInRangeFlag AND DS_HMI.b1000_00_AutoModeOnOffPB AND bInternalInput_b003_00_ChillerSelectorOnOff;

// NETWORK 6
DS_Output.i103_04_ChillerSelectorOnOffIndicator.0 := TRUE AND bInternalInput_b003_00_ChillerSelectorOnOff;
END_ACTION

ACTION FixOutput_LD:
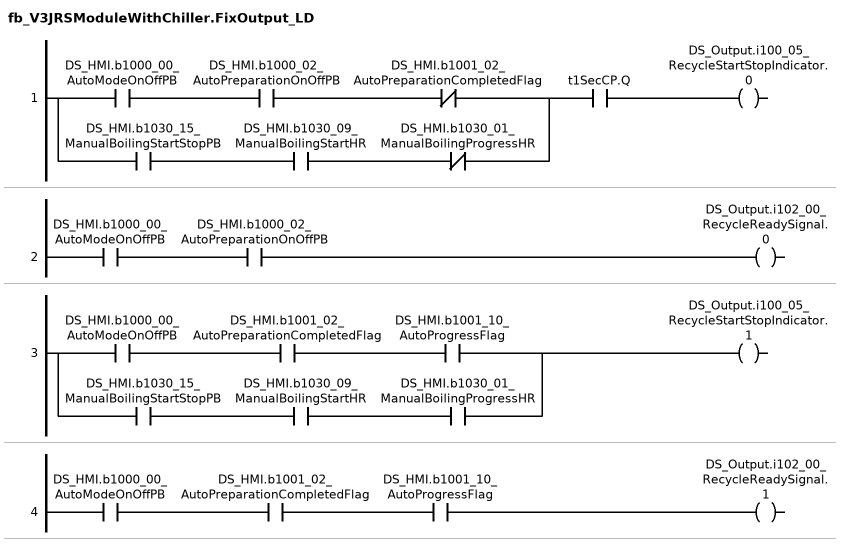
// NETWORK 1
DS_Output.i100_05_RecycleStartStopIndicator.0 := (DS_HMI.b1000_00_AutoModeOnOffPB AND DS_HMI.b1000_02_AutoPreparationOnOffPB AND NOT DS_HMI.b1001_02_AutoPreparationCompletedFlag OR DS_HMI.b1030_15_ManualBoilingStartStopPB AND DS_HMI.b1030_09_ManualBoilingStartHR AND NOT DS_HMI.b1030_01_ManualBoilingProgressHR) AND t1SecCP.Q;

// NETWORK 2
DS_Output.i102_00_RecycleReadySignal.0 := DS_HMI.b1000_00_AutoModeOnOffPB AND DS_HMI.b1000_02_AutoPreparationOnOffPB;

// NETWORK 3
DS_Output.i100_05_RecycleStartStopIndicator.1 := DS_HMI.b1000_00_AutoModeOnOffPB AND DS_HMI.b1001_02_AutoPreparationCompletedFlag AND DS_HMI.b1001_10_AutoProgressFlag OR DS_HMI.b1030_15_ManualBoilingStartStopPB AND DS_HMI.b1030_09_ManualBoilingStartHR AND DS_HMI.b1030_01_ManualBoilingProgressHR;

// NETWORK 4
DS_Output.i102_00_RecycleReadySignal.1 := DS_HMI.b1000_00_AutoModeOnOffPB AND DS_HMI.b1001_02_AutoPreparationCompletedFlag AND DS_HMI.b1001_10_AutoProgressFlag;
END_ACTION

ACTION HighLowLimitCtrl_ST:
(*Low Limit Ctrl*)
IF DS_HMI.iD490_ManualBoilCycleSV < 1 THEN
DS_HMI.iD490_ManualBoilCycleSV := 1;
END_IF

IF DS_HMI.iD200_AutoBoilProcessTimeSV_Min < 30 THEN
DS_HMI.iD200_AutoBoilProcessTimeSV_Min := 30;
END_IF

IF DS_HMI.iD201_AutoBoilDownTimeSV_Min < 5 THEN
DS_HMI.iD201_AutoBoilDownTimeSV_Min := 5;
END_IF

IF DS_HMI.iD202_AutoBoilDistillatorDrainTimeSV_Sec < 5 THEN
DS_HMI.iD202_AutoBoilDistillatorDrainTimeSV_Sec := 5;
END_IF

IF DS_HMI.iD203_AutoBoilSludgeDrainTimeSV_Sec < 5 THEN
DS_HMI.iD203_AutoBoilSludgeDrainTimeSV_Sec := 5;
END_IF

IF DS_HMI.iD210_ManualBoilDownTimeSV_Min < 5 THEN
DS_HMI.iD210_ManualBoilDownTimeSV_Min := 5;
END_IF

IF DS_HMI.iD211_ManualBoilSludgeCoolingTimeSV_Min < 1 THEN
DS_HMI.iD211_ManualBoilSludgeCoolingTimeSV_Min := 1;
END_IF

IF DS_HMI.iD212_ManualBoilSludgeDrainSV_Sec < 5 THEN
DS_HMI.iD212_ManualBoilSludgeDrainSV_Sec := 5;
END_IF




(*High LImit Ctrl*)
IF DS_HMI.iD490_ManualBoilCycleSV > 99 THEN
DS_HMI.iD490_ManualBoilCycleSV := 99;
END_IF

IF DS_HMI.iD200_AutoBoilProcessTimeSV_Min > 9999 THEN
DS_HMI.iD200_AutoBoilProcessTimeSV_Min := 9999;
END_IF

IF DS_HMI.iD201_AutoBoilDownTimeSV_Min > 9999 THEN
DS_HMI.iD201_AutoBoilDownTimeSV_Min := 9999;
END_IF

IF DS_HMI.iD202_AutoBoilDistillatorDrainTimeSV_Sec > 300 THEN
DS_HMI.iD202_AutoBoilDistillatorDrainTimeSV_Sec := 300;
END_IF

IF DS_HMI.iD203_AutoBoilSludgeDrainTimeSV_Sec > 300 THEN
DS_HMI.iD203_AutoBoilSludgeDrainTimeSV_Sec := 300;
END_IF

IF DS_HMI.iD210_ManualBoilDownTimeSV_Min > 99 THEN
DS_HMI.iD210_ManualBoilDownTimeSV_Min := 99;
END_IF

IF DS_HMI.iD211_ManualBoilSludgeCoolingTimeSV_Min > 9999 THEN
DS_HMI.iD211_ManualBoilSludgeCoolingTimeSV_Min := 9999;
END_IF

IF DS_HMI.iD212_ManualBoilSludgeDrainSV_Sec > 300 THEN
DS_HMI.iD212_ManualBoilSludgeDrainSV_Sec := 300;
END_IF
END_ACTION

ACTION JRSMachineServiceCtrl_LD:
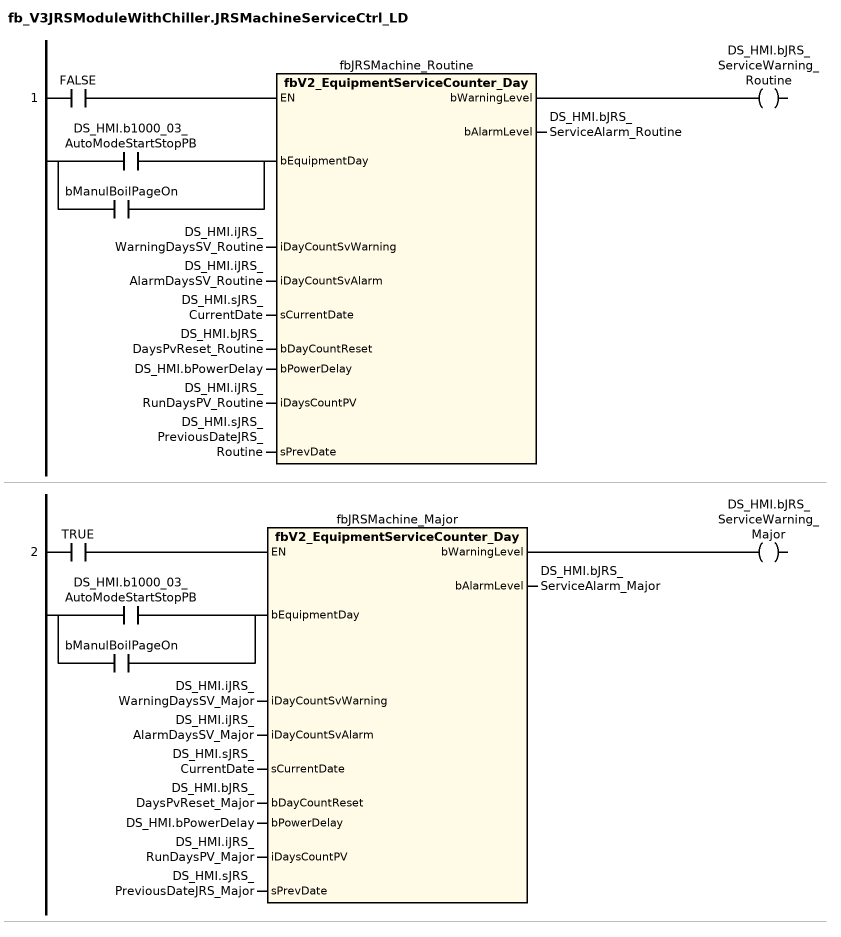
// NETWORK 1
IF FALSE THEN
    fbJRSMachine_Routine(
        bEquipmentDay := DS_HMI.b1000_03_AutoModeStartStopPB OR bManulBoilPageOn,
        iDayCountSvWarning := DS_HMI.iJRS_WarningDaysSV_Routine,
        iDayCountSvAlarm := DS_HMI.iJRS_AlarmDaysSV_Routine,
        sCurrentDate := DS_HMI.sJRS_CurrentDate,
        bDayCountReset := DS_HMI.bJRS_DaysPvReset_Routine,
        bPowerDelay := DS_HMI.bPowerDelay,
        iDaysCountPV := DS_HMI.iJRS_RunDaysPV_Routine,
        sPrevDate := DS_HMI.sJRS_PreviousDateJRS_Routine,
        bAlarmLevel => DS_HMI.bJRS_ServiceAlarm_Routine); // fbV2_EquipmentServiceCounter_Day
END_IF
DS_HMI.bJRS_ServiceWarning_Routine := fbJRSMachine_Routine.bWarningLevel;

// NETWORK 2
fbJRSMachine_Major(
    bEquipmentDay := DS_HMI.b1000_03_AutoModeStartStopPB OR bManulBoilPageOn,
    iDayCountSvWarning := DS_HMI.iJRS_WarningDaysSV_Major,
    iDayCountSvAlarm := DS_HMI.iJRS_AlarmDaysSV_Major,
    sCurrentDate := DS_HMI.sJRS_CurrentDate,
    bDayCountReset := DS_HMI.bJRS_DaysPvReset_Major,
    bPowerDelay := DS_HMI.bPowerDelay,
    iDaysCountPV := DS_HMI.iJRS_RunDaysPV_Major,
    sPrevDate := DS_HMI.sJRS_PreviousDateJRS_Major,
    bAlarmLevel => DS_HMI.bJRS_ServiceAlarm_Major); // fbV2_EquipmentServiceCounter_Day
DS_HMI.bJRS_ServiceWarning_Major := fbJRSMachine_Major.bWarningLevel;
END_ACTION

ACTION ManualBoilingCtrl_LD:
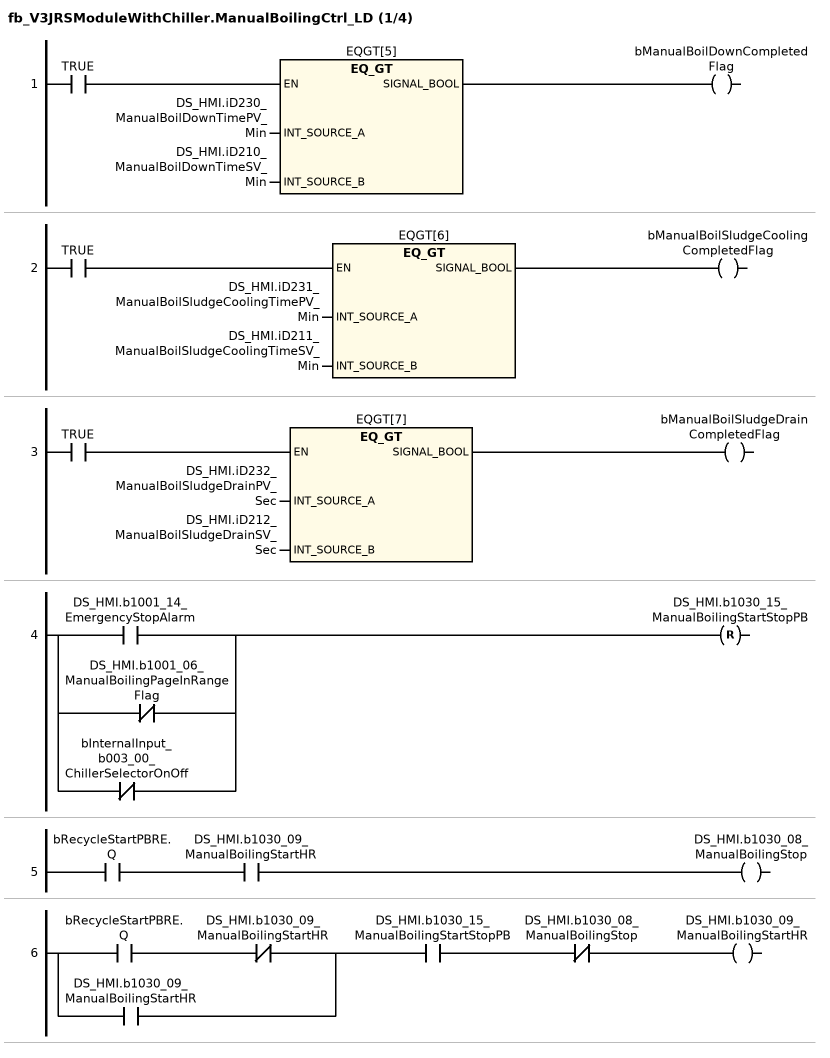
// NETWORK 1
EQGT[5](INT_SOURCE_A := DS_HMI.iD230_ManualBoilDownTimePV_Min, INT_SOURCE_B := DS_HMI.iD210_ManualBoilDownTimeSV_Min); // EQ_GT
bManualBoilDownCompletedFlag := EQGT[5].SIGNAL_BOOL;

// NETWORK 2
EQGT[6](INT_SOURCE_A := DS_HMI.iD231_ManualBoilSludgeCoolingTimePV_Min, INT_SOURCE_B := DS_HMI.iD211_ManualBoilSludgeCoolingTimeSV_Min); // EQ_GT
bManualBoilSludgeCoolingCompletedFlag := EQGT[6].SIGNAL_BOOL;

// NETWORK 3
EQGT[7](INT_SOURCE_A := DS_HMI.iD232_ManualBoilSludgeDrainPV_Sec, INT_SOURCE_B := DS_HMI.iD212_ManualBoilSludgeDrainSV_Sec); // EQ_GT
bManualBoilSludgeDrainCompletedFlag := EQGT[7].SIGNAL_BOOL;

// NETWORK 4
DS_HMI.b1030_15_ManualBoilingStartStopPB R= DS_HMI.b1001_14_EmergencyStopAlarm OR NOT DS_HMI.b1001_06_ManualBoilingPageInRangeFlag OR NOT bInternalInput_b003_00_ChillerSelectorOnOff;

// NETWORK 5
DS_HMI.b1030_08_ManualBoilingStop := bRecycleStartPBRE.Q AND DS_HMI.b1030_09_ManualBoilingStartHR;

// NETWORK 6
DS_HMI.b1030_09_ManualBoilingStartHR := (bRecycleStartPBRE.Q AND NOT DS_HMI.b1030_09_ManualBoilingStartHR OR DS_HMI.b1030_09_ManualBoilingStartHR) AND DS_HMI.b1030_15_ManualBoilingStartStopPB AND NOT DS_HMI.b1030_08_ManualBoilingStop;

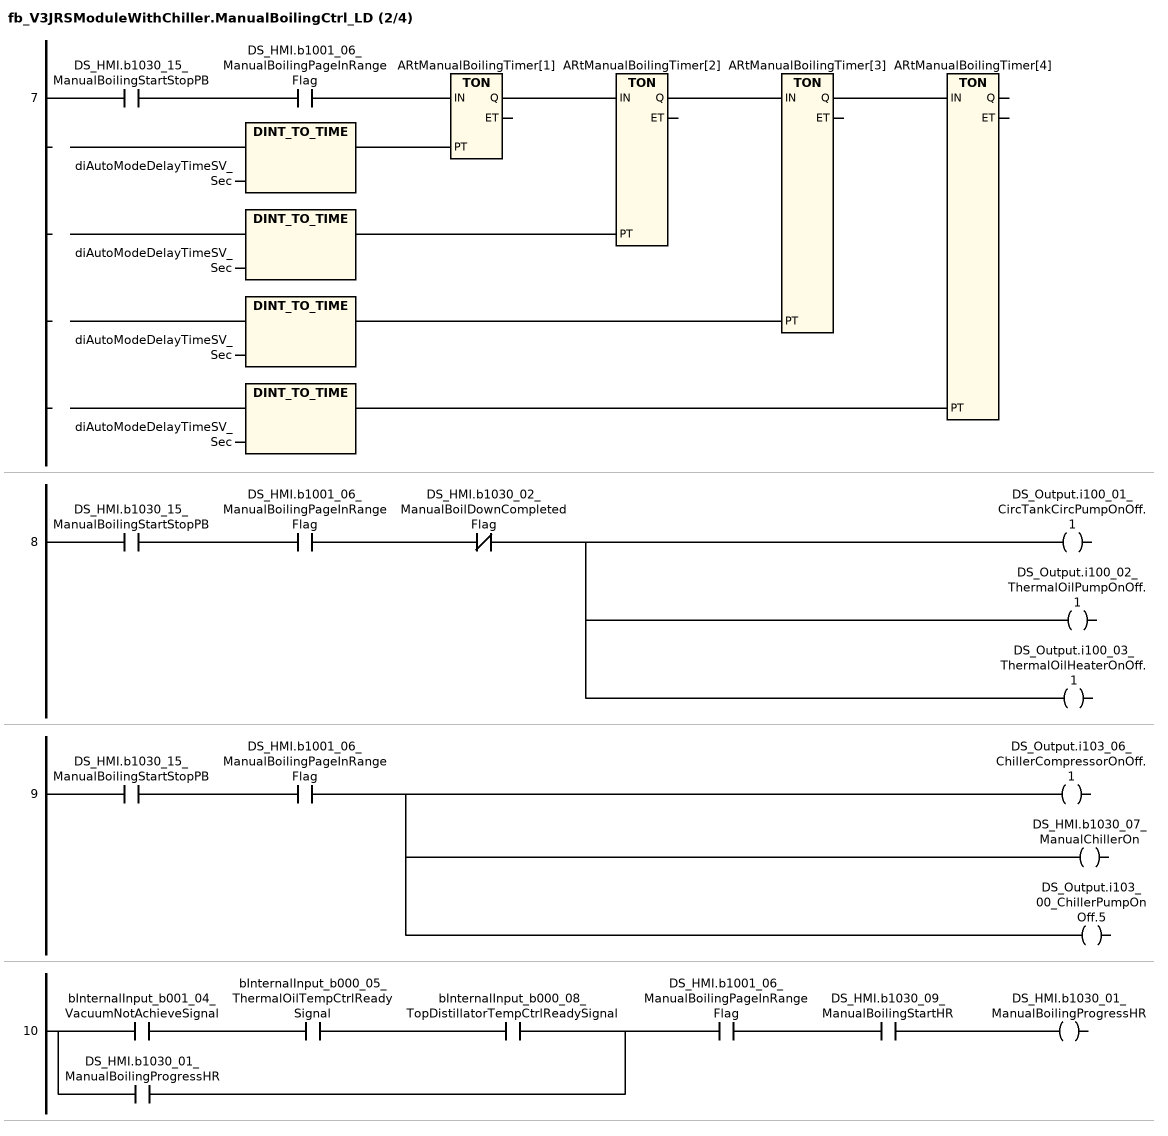
// NETWORK 7
ARtManualBoilingTimer[1](IN := DS_HMI.b1030_15_ManualBoilingStartStopPB AND DS_HMI.b1001_06_ManualBoilingPageInRangeFlag, PT := DINT_TO_TIME(diAutoModeDelayTimeSV_Sec)); // TON
ARtManualBoilingTimer[2](IN := ARtManualBoilingTimer[1].Q, PT := DINT_TO_TIME(diAutoModeDelayTimeSV_Sec)); // TON
ARtManualBoilingTimer[3](IN := ARtManualBoilingTimer[2].Q, PT := DINT_TO_TIME(diAutoModeDelayTimeSV_Sec)); // TON
ARtManualBoilingTimer[4](IN := ARtManualBoilingTimer[3].Q, PT := DINT_TO_TIME(diAutoModeDelayTimeSV_Sec)); // TON

// NETWORK 8
_w5 := DS_HMI.b1030_15_ManualBoilingStartStopPB AND DS_HMI.b1001_06_ManualBoilingPageInRangeFlag AND NOT DS_HMI.b1030_02_ManualBoilDownCompletedFlag;
DS_Output.i100_01_CircTankCircPumpOnOff.1 := _w5;
DS_Output.i100_02_ThermalOilPumpOnOff.1 := _w5;
DS_Output.i100_03_ThermalOilHeaterOnOff.1 := _w5;

// NETWORK 9
_w6 := DS_HMI.b1030_15_ManualBoilingStartStopPB AND DS_HMI.b1001_06_ManualBoilingPageInRangeFlag;
DS_Output.i103_06_ChillerCompressorOnOff.1 := _w6;
DS_HMI.b1030_07_ManualChillerOn := _w6;
DS_Output.i103_00_ChillerPumpOnOff.5 := _w6;

// NETWORK 10
DS_HMI.b1030_01_ManualBoilingProgressHR := (bInternalInput_b001_04_VacuumNotAchieveSignal AND bInternalInput_b000_05_ThermalOilTempCtrlReadySignal AND bInternalInput_b000_08_TopDistillatorTempCtrlReadySignal OR DS_HMI.b1030_01_ManualBoilingProgressHR) AND DS_HMI.b1001_06_ManualBoilingPageInRangeFlag AND DS_HMI.b1030_09_ManualBoilingStartHR;

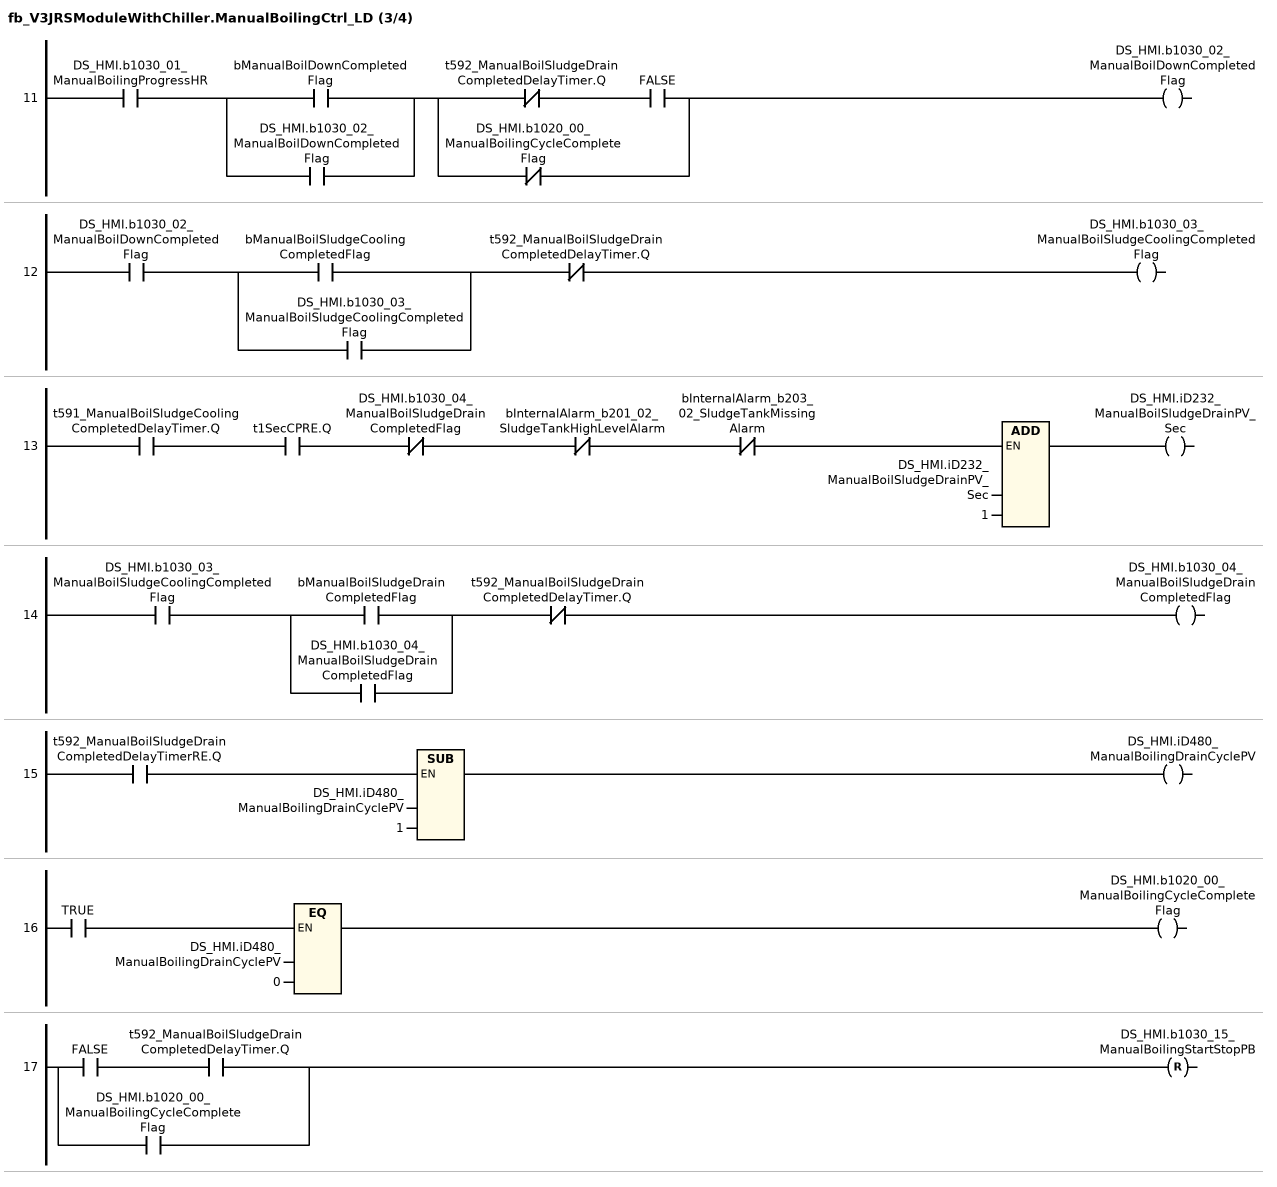
// NETWORK 11
DS_HMI.b1030_02_ManualBoilDownCompletedFlag := DS_HMI.b1030_01_ManualBoilingProgressHR AND (bManualBoilDownCompletedFlag OR DS_HMI.b1030_02_ManualBoilDownCompletedFlag) AND (NOT t592_ManualBoilSludgeDrainCompletedDelayTimer.Q AND FALSE OR NOT DS_HMI.b1020_00_ManualBoilingCycleCompleteFlag);

// NETWORK 12
DS_HMI.b1030_03_ManualBoilSludgeCoolingCompletedFlag := (DS_HMI.b1030_02_ManualBoilDownCompletedFlag AND (bManualBoilSludgeCoolingCompletedFlag OR DS_HMI.b1030_03_ManualBoilSludgeCoolingCompletedFlag)) AND NOT t592_ManualBoilSludgeDrainCompletedDelayTimer.Q;

// NETWORK 13
IF t591_ManualBoilSludgeCoolingCompletedDelayTimer.Q AND t1SecCPRE.Q AND NOT DS_HMI.b1030_04_ManualBoilSludgeDrainCompletedFlag AND NOT bInternalAlarm_b201_02_SludgeTankHighLevelAlarm AND NOT bInternalAlarm_b203_02_SludgeTankMissingAlarm THEN
    _w7 := DS_HMI.iD232_ManualBoilSludgeDrainPV_Sec + 1;
END_IF
DS_HMI.iD232_ManualBoilSludgeDrainPV_Sec := _w7;

// NETWORK 14
DS_HMI.b1030_04_ManualBoilSludgeDrainCompletedFlag := (DS_HMI.b1030_03_ManualBoilSludgeCoolingCompletedFlag AND (bManualBoilSludgeDrainCompletedFlag OR DS_HMI.b1030_04_ManualBoilSludgeDrainCompletedFlag)) AND NOT t592_ManualBoilSludgeDrainCompletedDelayTimer.Q;

// NETWORK 15
IF t592_ManualBoilSludgeDrainCompletedDelayTimerRE.Q THEN _w8 := DS_HMI.iD480_ManualBoilingDrainCyclePV - 1; END_IF
DS_HMI.iD480_ManualBoilingDrainCyclePV := _w8;

// NETWORK 16
DS_HMI.b1020_00_ManualBoilingCycleCompleteFlag := DS_HMI.iD480_ManualBoilingDrainCyclePV = 0;

// NETWORK 17
DS_HMI.b1030_15_ManualBoilingStartStopPB R= FALSE AND t592_ManualBoilSludgeDrainCompletedDelayTimer.Q OR DS_HMI.b1020_00_ManualBoilingCycleCompleteFlag;

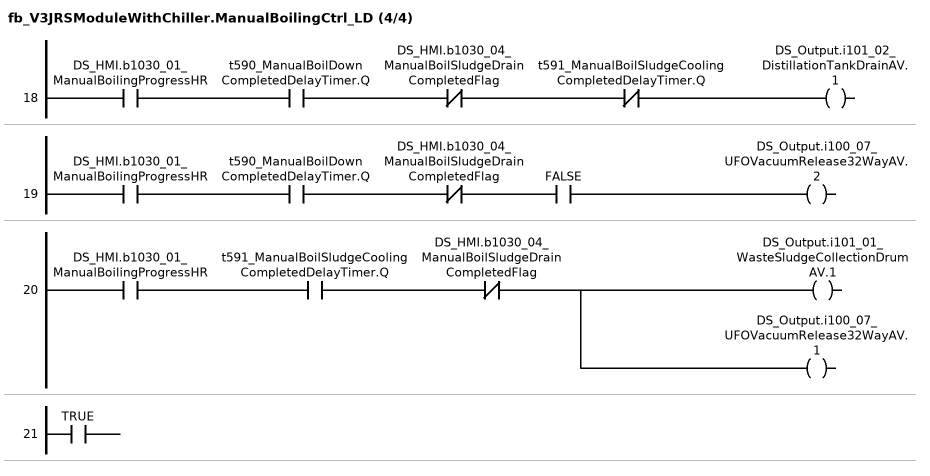
// NETWORK 18
DS_Output.i101_02_DistillationTankDrainAV.1 := DS_HMI.b1030_01_ManualBoilingProgressHR AND t590_ManualBoilDownCompletedDelayTimer.Q AND NOT DS_HMI.b1030_04_ManualBoilSludgeDrainCompletedFlag AND NOT t591_ManualBoilSludgeCoolingCompletedDelayTimer.Q;

// NETWORK 19
DS_Output.i100_07_UFOVacuumRelease32WayAV.2 := DS_HMI.b1030_01_ManualBoilingProgressHR AND t590_ManualBoilDownCompletedDelayTimer.Q AND NOT DS_HMI.b1030_04_ManualBoilSludgeDrainCompletedFlag AND FALSE;

// NETWORK 20
_w9 := DS_HMI.b1030_01_ManualBoilingProgressHR AND t591_ManualBoilSludgeCoolingCompletedDelayTimer.Q AND NOT DS_HMI.b1030_04_ManualBoilSludgeDrainCompletedFlag;
DS_Output.i101_01_WasteSludgeCollectionDrumAV.1 := _w9;
DS_Output.i100_07_UFOVacuumRelease32WayAV.1 := _w9;

// NETWORK 21
END_ACTION

ACTION ManualBoilingCtrl_ST:
	(*Timer*)
	t590_ManualBoilDownCompletedDelayTimer(IN:=DS_HMI.b1030_02_ManualBoilDownCompletedFlag , PT:=t#1s , Q=> , ET=> );
	t591_ManualBoilSludgeCoolingCompletedDelayTimer(IN:=DS_HMI.b1030_03_ManualBoilSludgeCoolingCompletedFlag , PT:=t#1s , Q=> , ET=> );
	t592_ManualBoilSludgeDrainCompletedDelayTimer(IN:=DS_HMI.b1030_04_ManualBoilSludgeDrainCompletedFlag , PT:=t#1s , Q=> , ET=> );

	(*R_TRIG*)
	t592_ManualBoilSludgeDrainCompletedDelayTimerRE(CLK:=t592_ManualBoilSludgeDrainCompletedDelayTimer.Q , Q=> );
	bManualBoilSludgeDrainCompletedRE(CLK:=DS_HMI.b1030_04_ManualBoilSludgeDrainCompletedFlag , Q=> );


	(*ManualBoiling Boil Process Time Counting*)
	IF DS_HMI.b1030_01_ManualBoilingProgressHR
	AND t1SecCPRE.Q
	THEN

		IF NOT DS_HMI.b1030_02_ManualBoilDownCompletedFlag THEN

			DS_HMI.iD235_ManualBoilDownTimePV_Sec := DS_HMI.iD235_ManualBoilDownTimePV_Sec + 1;
	
			IF DS_HMI.iD235_ManualBoilDownTimePV_Sec > 59 THEN
				DS_HMI.iD230_ManualBoilDownTimePV_Min := DS_HMI.iD230_ManualBoilDownTimePV_Min + 1;
				DS_HMI.iD235_ManualBoilDownTimePV_Sec := 0;
			END_IF

		END_IF

	END_IF

	(*ManualBoiling Boil Down Time Counting*)

	IF t590_ManualBoilDownCompletedDelayTimer.Q
	AND t1SecCPRE.Q
	THEN

		IF NOT DS_HMI.b1030_03_ManualBoilSludgeCoolingCompletedFlag THEN

			DS_HMI.iD236_ManualBoilSludgeCoolingTimePV_Sec := DS_HMI.iD236_ManualBoilSludgeCoolingTimePV_Sec + 1;

			IF DS_HMI.iD236_ManualBoilSludgeCoolingTimePV_Sec > 59 THEN
				DS_HMI.iD231_ManualBoilSludgeCoolingTimePV_Min := DS_HMI.iD231_ManualBoilSludgeCoolingTimePV_Min + 1;
				DS_HMI.iD236_ManualBoilSludgeCoolingTimePV_Sec := 0;
			END_IF

		END_IF

	END_IF

	(*Manual Boiling Reset*)
	IF NOT DS_HMI.b1030_15_ManualBoilingStartStopPB THEN
		DS_HMI.iD230_ManualBoilDownTimePV_Min						:= 0;
		DS_HMI.iD231_ManualBoilSludgeCoolingTimePV_Min				:= 0;
		DS_HMI.iD232_ManualBoilSludgeDrainPV_Sec					:= 0;
		DS_HMI.iD480_ManualBoilingDrainCyclePV						:= DS_HMI.iD490_ManualBoilCycleSV;

	END_IF



	IF bManualBoilSludgeDrainCompletedRE.Q OR  DS_HMI.b1020_00_ManualBoilingCycleCompleteFlag THEN
	
		DS_HMI.iD230_ManualBoilDownTimePV_Min						:= 0;
		DS_HMI.iD231_ManualBoilSludgeCoolingTimePV_Min				:= 0;
		DS_HMI.iD232_ManualBoilSludgeDrainPV_Sec					:= 0;
		DS_HMI.iD235_ManualBoilDownTimePV_Sec						:= 0;
		DS_HMI.iD236_ManualBoilSludgeCoolingTimePV_Sec				:= 0;

	END_IF
END_ACTION

ACTION ManualCtrl_ST:
	(*Manual Page In Range*)
	IF (	DS_HMI.iD0_HMICurrentPage > 19 		AND 	DS_HMI.iD0_HMICurrentPage < 41)
	OR	DS_HMI.iD0_HMICurrentPage = 2
	OR	DS_HMI.iD0_HMICurrentPage = 61
	OR	DS_HMI.iD0_HMICurrentPage = 63
	OR	DS_HMI.iD0_HMICurrentPage = 100
	OR	DS_HMI.iD0_HMICurrentPage = 101
	OR	DS_HMI.iD0_HMICurrentPage = 103 	THEN
		DS_HMI.b1001_09_ManualPageInRangeFlag := TRUE;
	ELSE
		DS_HMI.b1001_09_ManualPageInRangeFlag := FALSE;
	END_IF


	(*Manual Boiling Page In Range*)
	IF (	DS_HMI.iD0_HMICurrentPage > 99 		AND 	DS_HMI.iD0_HMICurrentPage < 102)
	OR	DS_HMI.iD0_HMICurrentPage = 22 		THEN
		DS_HMI.b1001_06_ManualBoilingPageInRangeFlag := TRUE;
	ELSE
		DS_HMI.b1001_06_ManualBoilingPageInRangeFlag := FALSE;
	END_IF



	IF NOT DS_HMI.b1001_09_ManualPageInRangeFlag OR DS_HMI.b1001_14_EmergencyStopAlarm THEN
		DS_Output.i100_00_FreshHCTankCircPumpOnOff.15			:= FALSE;
		DS_Output.i100_01_CircTankCircPumpOnOff.15				:= FALSE;
		DS_Output.i100_02_ThermalOilPumpOnOff.15				:= FALSE;
		DS_Output.i100_03_ThermalOilHeaterOnOff.15				:= FALSE;
		DS_Output.i100_04_Buzzer.15								:= FALSE;
		DS_Output.i100_05_RecycleStartStopIndicator.15				:= FALSE;
		DS_Output.i100_06_Reserved.15							:= FALSE;
		DS_Output.i100_07_UFOVacuumRelease32WayAV.15		:= FALSE;

		DS_Output.i101_00_CondenserTankVacuumReleaseAV.15	:= FALSE;
		DS_Output.i101_01_WasteSludgeCollectionDrumAV.15		:= FALSE;
		DS_Output.i101_02_DistillationTankDrainAV.15				:= FALSE;
		DS_Output.i101_03_EconomizerAV.15						:= FALSE;
		DS_Output.i101_04_Reserved.15							:= FALSE;
		DS_Output.i101_05_Reserved.15							:= FALSE;
		DS_Output.i101_06_VaporGenerationAV.15					:= FALSE;
		DS_Output.i101_07_VacuumSharingAV.15					:= FALSE;

		DS_Output.i102_00_RecycleReadySignal.15					:= FALSE;
		DS_Output.i102_01_VaporNotAvailableForRequestSignal.15	:= FALSE;
		DS_Output.i102_02_ToMainMachineSignal3.15				:= FALSE;
		DS_Output.i102_03_ToMainMachineSignal4.15				:= FALSE;
		DS_Output.i102_04_ToMainMachineSignal5.15				:= FALSE;
		DS_Output.i102_05_Reserved.15							:= FALSE;
		DS_Output.i102_06_Reserved.15							:= FALSE;
		DS_Output.i102_07_Reserved.15							:= FALSE;

		DS_Output.i103_00_ChillerPumpOnOff.15					:= FALSE;
		DS_Output.i103_01_Reserved.15							:= FALSE;
		DS_Output.i103_02_Reserved.15							:= FALSE;
		DS_Output.i103_03_Reserved.15							:= FALSE;
		DS_Output.i103_04_ChillerSelectorOnOffIndicator.15			:= FALSE;
		DS_Output.i103_05_ChillerReadySignal.15					:= FALSE;
		DS_Output.i103_06_ChillerCompressorOnOff.15				:= FALSE;
		DS_Output.i103_07_Reserved.15							:= FALSE;
	END_IF

	IF NOT bInternalInput_b003_00_ChillerSelectorOnOff THEN
		DS_Output.i103_06_ChillerCompressorOnOff.15				:= FALSE;
	END_IF
END_ACTION

ACTION MessageDisplayCtrl_ST:
	IF  NOT DS_HMI.b1001_15_AlarmOccur THEN

		IF NOT 		DS_HMI.b1000_00_AutoModeOnOffPB THEN

			DS_HMI.iD100_MessageDisplay := 0;
			DS_HMI.sD100_MessageDisplay := 'Machine Idle';

(*		ELSIF 		DS_HMI.b1000_00_AutoModeOnOffPB
		AND 		DS_HMI.b1000_01_AutoOriginOnOffPB
		AND NOT 	DS_HMI.b1001_01_AutoOriginCompletedFlag THEN

			DS_HMI.iD100_MessageDisplay := 1;
			DS_HMI.sD100_MessageDisplay := 'Auto Origin In Progress...';
*)
		ELSIF 		DS_HMI.b1000_00_AutoModeOnOffPB
		AND 		DS_HMI.b1000_02_AutoPreparationOnOffPB
		AND NOT 	DS_HMI.b1001_02_AutoPreparationCompletedFlag THEN

			DS_HMI.iD100_MessageDisplay := 2;
			DS_HMI.sD100_MessageDisplay := 'Auto Preparation In Progress...';

		ELSIF 		DS_HMI.b1000_00_AutoModeOnOffPB
(*		AND 		DS_HMI.b1001_01_AutoOriginCompletedFlag*)
		AND 		DS_HMI.b1000_02_AutoPreparationOnOffPB
		AND 		DS_HMI.b1001_02_AutoPreparationCompletedFlag THEN

			DS_HMI.iD100_MessageDisplay := 3;
			DS_HMI.sD100_MessageDisplay := 'Machine Ready, Press "Start" for Operation';

		ELSIF 		DS_HMI.b1000_00_AutoModeOnOffPB
(*		AND 		DS_HMI.b1001_01_AutoOriginCompletedFlag*)
		AND 		DS_HMI.b1001_02_AutoPreparationCompletedFlag
		AND 		DS_HMI.b1001_10_AutoProgressFlag
		AND NOT 	DS_HMI.b1000_05_AutoCycleStopPB THEN

			DS_HMI.iD100_MessageDisplay := 4;
			DS_HMI.sD100_MessageDisplay := 'Machine Operation...';

		ELSIF 		DS_HMI.b1000_00_AutoModeOnOffPB
(*		AND 		DS_HMI.b1001_01_AutoOriginCompletedFlag*)
		AND 		DS_HMI.b1001_02_AutoPreparationCompletedFlag
		AND 		DS_HMI.b1001_10_AutoProgressFlag
		AND 		DS_HMI.b1000_05_AutoCycleStopPB THEN

			DS_HMI.iD100_MessageDisplay := 5;
			DS_HMI.sD100_MessageDisplay := 'Auto Cycle Stop...';

		END_IF

	ELSE
		DS_HMI.iD100_MessageDisplay := 6;
			DS_HMI.sD100_MessageDisplay := 'Alarm Occured, Please check Alarm Page for more detail';

	END_IF
END_ACTION

ACTION Other_LD:
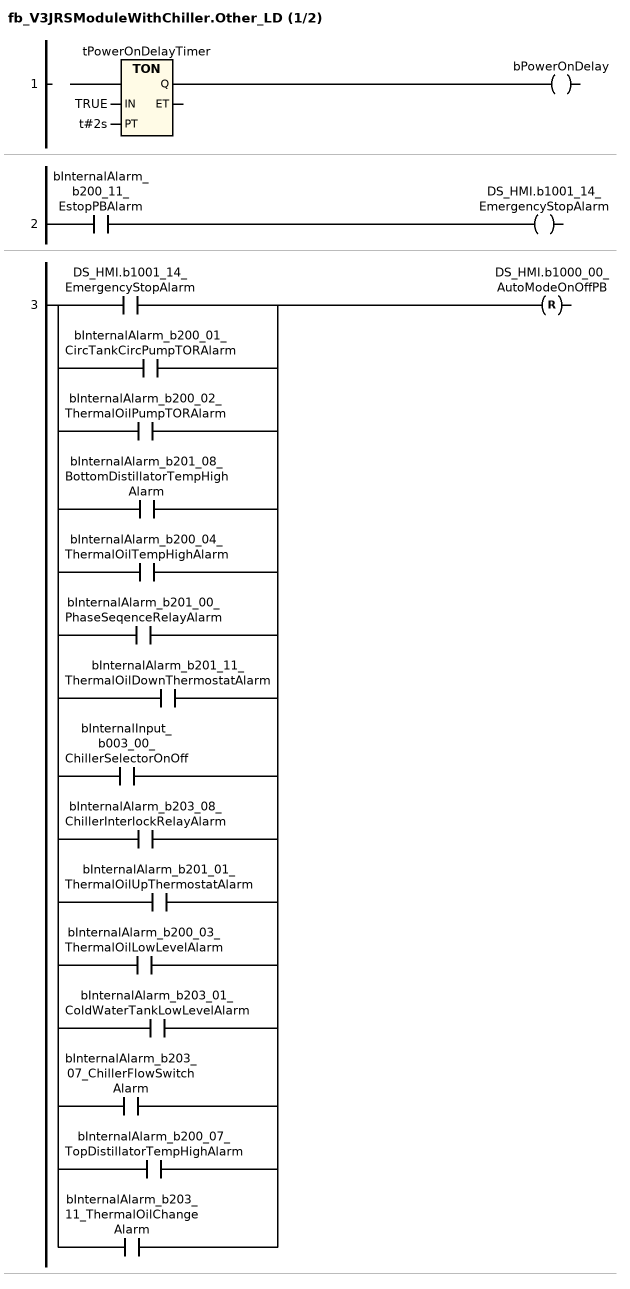
// NETWORK 1
tPowerOnDelayTimer(IN := TRUE, PT := t#2s); // TON
bPowerOnDelay := tPowerOnDelayTimer.Q;

// NETWORK 2
DS_HMI.b1001_14_EmergencyStopAlarm := bInternalAlarm_b200_11_EstopPBAlarm;

// NETWORK 3
DS_HMI.b1000_00_AutoModeOnOffPB R= DS_HMI.b1001_14_EmergencyStopAlarm OR bInternalAlarm_b200_01_CircTankCircPumpTORAlarm OR bInternalAlarm_b200_02_ThermalOilPumpTORAlarm OR bInternalAlarm_b201_08_BottomDistillatorTempHighAlarm OR bInternalAlarm_b200_04_ThermalOilTempHighAlarm OR bInternalAlarm_b201_00_PhaseSeqenceRelayAlarm OR bInternalAlarm_b201_11_ThermalOilDownThermostatAlarm OR bInternalInput_b003_00_ChillerSelectorOnOff OR bInternalAlarm_b203_08_ChillerInterlockRelayAlarm OR bInternalAlarm_b201_01_ThermalOilUpThermostatAlarm OR bInternalAlarm_b200_03_ThermalOilLowLevelAlarm OR bInternalAlarm_b203_01_ColdWaterTankLowLevelAlarm OR bInternalAlarm_b203_07_ChillerFlowSwitchAlarm OR bInternalAlarm_b200_07_TopDistillatorTempHighAlarm OR bInternalAlarm_b203_11_ThermalOilChangeAlarm;

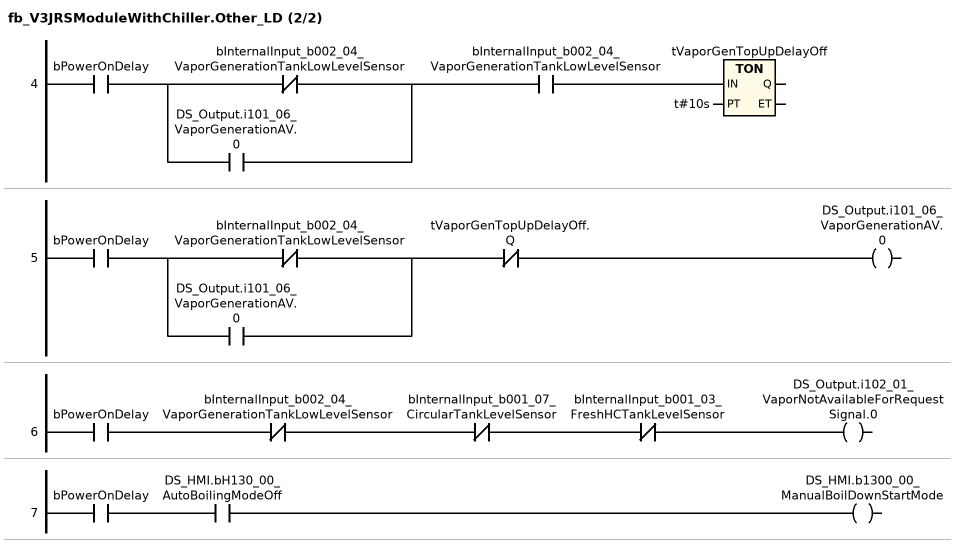
// NETWORK 4
tVaporGenTopUpDelayOff(IN := (bPowerOnDelay AND (NOT bInternalInput_b002_04_VaporGenerationTankLowLevelSensor OR DS_Output.i101_06_VaporGenerationAV.0)) AND bInternalInput_b002_04_VaporGenerationTankLowLevelSensor, PT := t#10s); // TON

// NETWORK 5
DS_Output.i101_06_VaporGenerationAV.0 := (bPowerOnDelay AND (NOT bInternalInput_b002_04_VaporGenerationTankLowLevelSensor OR DS_Output.i101_06_VaporGenerationAV.0)) AND NOT tVaporGenTopUpDelayOff.Q;

// NETWORK 6
DS_Output.i102_01_VaporNotAvailableForRequestSignal.0 := bPowerOnDelay AND NOT bInternalInput_b002_04_VaporGenerationTankLowLevelSensor AND NOT bInternalInput_b001_07_CircularTankLevelSensor AND NOT bInternalInput_b001_03_FreshHCTankLevelSensor;

// NETWORK 7
DS_HMI.b1300_00_ManualBoilDownStartMode := bPowerOnDelay AND DS_HMI.bH130_00_AutoBoilingModeOff;
END_ACTION

ACTION Other_ST:
	(*Map Alarm into Word so that can generate Alarm Occur Bit*)
	AriAlarmFlag[1].0 := bInternalAlarm_b200_00_FreshHCTankCircPumpTORAlarm ;
	AriAlarmFlag[1].1 := bInternalAlarm_b200_01_CircTankCircPumpTORAlarm ;
	AriAlarmFlag[1].2 := bInternalAlarm_b200_02_ThermalOilPumpTORAlarm ;
	AriAlarmFlag[1].3 := bInternalAlarm_b200_03_ThermalOilLowLevelAlarm ;
	AriAlarmFlag[1].4 := bInternalAlarm_b200_04_ThermalOilTempHighAlarm ;
	AriAlarmFlag[1].5 := bInternalAlarm_b200_05_ThermalOilTempNotReadyAlarm ;
	AriAlarmFlag[1].6 := bInternalAlarm_b200_06_ThermalOilHeaterOnOffAlarm ;
	AriAlarmFlag[1].7 := bInternalAlarm_b200_07_TopDistillatorTempHighAlarm ;
	AriAlarmFlag[1].8 := bInternalAlarm_b200_08_TopDistillatorTempNotReadyAlarm ;
	AriAlarmFlag[1].9 := bInternalAlarm_b200_09_TopDistillatorHeaterOnOffAlarm ;
	AriAlarmFlag[1].10 := bInternalAlarm_b200_10_RecycleStartStopPBAlarm ;
	AriAlarmFlag[1].11 := bInternalAlarm_b200_11_EstopPBAlarm ;
	
	AriAlarmFlag[2].0 := bInternalAlarm_b201_00_PhaseSeqenceRelayAlarm ;
	AriAlarmFlag[2].1 := bInternalAlarm_b201_01_ThermalOilUpThermostatAlarm ;
	AriAlarmFlag[2].2 := bInternalAlarm_b201_02_SludgeTankHighLevelAlarm ;
	AriAlarmFlag[2].3 := bInternalAlarm_b201_03_FreshHCTankLowLevelAlarm ;
	AriAlarmFlag[2].4 := bInternalAlarm_b201_04_VacuumNotAchieveAlarm ;
	AriAlarmFlag[2].5 := bInternalAlarm_b201_05_IncomingCDALowPressureAlarm ;
	AriAlarmFlag[2].6 := bInternalAlarm_b201_06_CoolingWaterLowFlowAlarm ;
	AriAlarmFlag[2].7 := bInternalAlarm_b201_07_CircularTankLowLevelAlarm ;
	AriAlarmFlag[2].8 := bInternalAlarm_b201_08_BottomDistillatorTempHighAlarm ;
	AriAlarmFlag[2].9 := bInternalAlarm_b201_09_BottomDistillatorTempNotReadyAlarm ;
	AriAlarmFlag[2].10 := bInternalAlarm_b201_10_BottomDistillatorHeaterOnOffAlarm ;
	AriAlarmFlag[2].11 := bInternalAlarm_b201_11_ThermalOilDownThermostatAlarm ;
	AriAlarmFlag[2].12 := bInternalAlarm_b201_12_ThermalOilMidThermostatAlarm ;

	AriAlarmFlag[3].0 := bInternalAlarm_b202_00_VaporGenerationTempHighAlarm ;
	AriAlarmFlag[3].1 := bInternalAlarm_b202_01_VaporGenerationTempNotReadyAlarm ;
	AriAlarmFlag[3].2 := bInternalAlarm_b202_02_VaporGenerationHeaterOnOffAlarm ;
	AriAlarmFlag[3].3 := bInternalAlarm_b202_03_WasteCollectionTankLowLevelAlarm ;
	AriAlarmFlag[3].4 := bInternalAlarm_b202_04_VaporGenerationTankLowLevelAlarm ;
	AriAlarmFlag[3].5 := bInternalAlarm_b202_05_HCPurgingAV3_1Alarm ;
	AriAlarmFlag[3].6 := bInternalAlarm_b202_06_MainMachineWasteTankLowLevelAlarm ;
	AriAlarmFlag[3].7 := bInternalAlarm_b202_07_MainMachineWasteTankHighLevelAlarm ;
	AriAlarmFlag[3].8 := bInternalAlarm_b202_08_ReservedAlarm ;
	AriAlarmFlag[3].9 := bInternalAlarm_b202_09_ReservedAlarm ;
	AriAlarmFlag[3].10 := bInternalAlarm_b202_10_ReservedAlarm ;
	AriAlarmFlag[3].11 := bInternalAlarm_b202_11_ReservedAlarm ;
	
	AriAlarmFlag[4].0 := bInternalAlarm_b203_00_ChillerSelectorOnOffAlarm ;
	AriAlarmFlag[4].1 := bInternalAlarm_b203_01_ColdWaterTankLowLevelAlarm ;
	AriAlarmFlag[4].2 := bInternalAlarm_b203_02_SludgeTankMissingAlarm ;
	AriAlarmFlag[4].3 := bInternalAlarm_b203_03_ColdWaterTankTempHighAlarm ;
	AriAlarmFlag[4].4 := bInternalAlarm_b203_04_ColdWaterTankTempNotReadyAlarm ;
	AriAlarmFlag[4].5 := bInternalAlarm_b203_05_ColdWaterTankHeaterOnOffAlarm ;
	AriAlarmFlag[4].6 := bInternalAlarm_b203_06_ChillerPumpTORAlarm ;
	AriAlarmFlag[4].7 := bInternalAlarm_b203_07_ChillerFlowSwitchAlarm ;
	AriAlarmFlag[4].8 := bInternalAlarm_b203_08_ChillerInterlockRelayAlarm ;
	AriAlarmFlag[4].9 := bInternalAlarm_b203_09_ReservedAlarm ;
	AriAlarmFlag[4].10 := bInternalAlarm_b203_10_ThermalOilChangeWarning ;
	AriAlarmFlag[4].11 := bInternalAlarm_b203_11_ThermalOilChangeAlarm ;
	
	
	IF AriAlarmFlag[1] <> 0
	OR AriAlarmFlag[2] <> 0
	OR AriAlarmFlag[3] <> 0
	OR AriAlarmFlag[4] <> 0
	THEN
	DS_HMI.b1001_15_AlarmOccur := TRUE;
	ELSE
	DS_HMI.b1001_15_AlarmOccur := FALSE;
	END_IF
END_ACTION

ACTION OutputCtrl_LD:
